// Functions/Keypoint Features/F_VN_FindReferenceKeyPointsInImageAKAZE

	{attribute 'TcIecLibraryType'}
	{attribute 'external_name' := 'F_VN_FindReferenceKeyPointsInImageAKAZE_GUID_BDEC472E_8EBA_B1D3_501C_E84D71D3DFEF'}
	(* Searches a reference image, represented by its AKAZE keypoints and corresponding descriptors, in a given source image (uses the default TcVnParamsAKAZE parameters). *)
	FUNCTION F_VN_FindReferenceKeyPointsInImageAKAZE : HRESULT
	VAR_INPUT
		ipSrcImage	:	ITcVnImage;	(* Source image *)
		ipRefKeyPoints	:	ITcVnContainer;	(* KeyPoints of the reference image, e.g. computed with F_VN_KeyPointsAndDescriptorsAKAZE (ContainerType_Vector_TcVnKeyPoint) *)
		ipRefDescriptors	:	ITcVnImage;	(* Descriptors of the reference image KeyPoints, e.g. computed with F_VN_KeyPointsAndDescriptorsAKAZE *)
		nRefImageWidth	:	UDINT;	(* Width of the reference image in pixels *)
		nRefImageHeight	:	UDINT;	(* Height of the reference image in pixels *)
		ipEdgePoints	:	REFERENCE TO ITcVnContainer;	(* Returns a container with the 4 edge points of the reference image transformed into ipSrcImage coordinates (ContainerType_Vector_TcVnPoint2_REAL) *)
		fMaxDist	:	REAL;	(* Maximum allowed descriptor distance (-1 disables this filter criterion) *)
		fMaxKnnRatio	:	REAL;	(* Maximum allowed distance ratio between first and second best match ([0..1], -1 disables this filter criterion) *)
		hrPrev	:	HRESULT;	(* HRESULT indicating the result of previous operations (If SUCCEEDED(hrPrev) equals false, no operation is executed.) *)
	END_VAR
	VAR_OUTPUT
		aPerspectiveTransform	:	TcVnMatrix3x3_LREAL;	(* Returns the perspective transformation matrix, which transforms the reference points to the source points *)
		nNumberOfGoodMatches	:	UDINT;	(* Return the number of good matches *)
		nNumberOfInliers	:	UDINT;	(* Return the number of inlier matches *)
	END_VAR

END_FUNCTION

// Functions/Keypoint Features/F_VN_KeyPointsAndDescriptorsAKAZE

	{attribute 'TcIecLibraryType'}
	{attribute 'external_name' := 'F_VN_KeyPointsAndDescriptorsAKAZE_GUID_3790B025_A52C_B22C_6EF2_34873295F067'}
	(* Detects keypoints and compute descriptors using the AKAZE method. *)
	FUNCTION F_VN_KeyPointsAndDescriptorsAKAZE : HRESULT
	VAR_INPUT
		ipSrcImage	:	ITcVnImage;	(* Source image *)
		ipKeyPoints	:	REFERENCE TO ITcVnContainer;	(* Returns a container which is filled with the keypoints (ContainerType_Vector_TcVnKeyPoint; Non-zero interface pointers are reused.) *)
		ipDescriptors	:	REFERENCE TO ITcVnImage;	(* Descriptor image (set to 0 if not required; 1 descriptor in each row; An appropriate image will be created if required.) *)
		hrPrev	:	HRESULT;	(* HRESULT indicating the result of previous operations (If SUCCEEDED(hrPrev) equals false, no operation is executed.) *)
	END_VAR

END_FUNCTION

// Functions/Keypoint Features/F_VN_FindReferenceKeyPointsInImageAKAZEExp

	{attribute 'TcIecLibraryType'}
	{attribute 'external_name' := 'F_VN_FindReferenceKeyPointsInImageAKAZEExp_GUID_5E4CFD0A_CE1D_BA8B_45D3_79DE9C5B1A21'}
	(* Searches a reference image, represented by its AKAZE keypoints and corresponding descriptors, in a given source image. (expert function) *)
	FUNCTION F_VN_FindReferenceKeyPointsInImageAKAZEExp : HRESULT
	VAR_INPUT
		ipSrcImage	:	ITcVnImage;	(* Source image *)
		ipRefKeyPoints	:	ITcVnContainer;	(* KeyPoints of the reference image, e.g. computed with F_VN_KeyPointsAndDescriptorsAKAZE (ContainerType_Vector_TcVnKeyPoint) *)
		ipRefDescriptors	:	ITcVnImage;	(* Descriptors of the reference image KeyPoints, e.g. computed with F_VN_KeyPointsAndDescriptorsAKAZE *)
		nRefImageWidth	:	UDINT;	(* Width of the reference image in pixels *)
		nRefImageHeight	:	UDINT;	(* Height of the reference image in pixels *)
		ipEdgePoints	:	REFERENCE TO ITcVnContainer;	(* Returns a container with the 4 edge points of the reference image transformed into ipSrcImage coordinates (ContainerType_Vector_TcVnPoint2_REAL) *)
		fMaxDist	:	REAL;	(* Maximum allowed descriptor distance (-1 disables this filter criterion) *)
		fMaxKnnRatio	:	REAL;	(* Maximum allowed distance ratio between first and second best match ([0..1], -1 disables this filter criterion) *)
		eNormType	:	ETcVnNormalizationType;	(* Normalization type used for descriptor matching *)
		ipSrcImageMask	:	ITcVnImage;	(* Mask to specify, where to look for keypoints in ipSrcImage (set to 0 if no mask required) *)
	END_VAR
	VAR_IN_OUT
		stAkazeParams	:	TcVnParamsAKAZE;	(* Parameters to configure the keypoint and descriptor computation for ipSrcImage (resulting descriptors must be compatible to ipRefDescriptors!) *)
	END_VAR
	VAR_INPUT
		eAlgorithm	:	ETcVnEstimationAlgorithm;	(* Estimation algorithm used for computing the perspective transformation between the two point sets *)
		fReprojThreshold	:	LREAL;	(* Maximum allowed reprojection error to treat a point pair as an inlier (only used if eAlgorithm is RANSAC, RHO) *)
		nMaxIterations	:	UDINT;	(* Maximum number of RANSAC iterations *)
		fConfidence	:	LREAL;	(* Confidence (0..1) *)
		hrPrev	:	HRESULT;	(* HRESULT indicating the result of previous operations (If SUCCEEDED(hrPrev) equals false, no operation is executed.) *)
	END_VAR
	VAR_OUTPUT
		aPerspectiveTransform	:	TcVnMatrix3x3_LREAL;	(* Returns the perspective transformation matrix, which transforms the reference points to the source points  *)
		nNumberOfGoodMatches	:	UDINT;	(* Return the number of good matches *)
		nNumberOfInliers	:	UDINT;	(* Return the number of inlier matches *)
	END_VAR

END_FUNCTION

// Functions/Keypoint Features/F_VN_FindReferenceKeyPointsInImageBRISK

	{attribute 'TcIecLibraryType'}
	{attribute 'external_name' := 'F_VN_FindReferenceKeyPointsInImageBRISK_GUID_C2D82A25_9CFE_BE26_6FAE_778E3D975A2B'}
	(* Searches a reference image, represented by its BRISK keypoints and corresponding descriptors, in a given source image (uses the default TcVnParamsBRISK parameters). *)
	FUNCTION F_VN_FindReferenceKeyPointsInImageBRISK : HRESULT
	VAR_INPUT
		ipSrcImage	:	ITcVnImage;	(* Source image *)
		ipRefKeyPoints	:	ITcVnContainer;	(* KeyPoints of the reference image, e.g. computed with F_VN_KeyPointsAndDescriptorsBRISK (ContainerType_Vector_TcVnKeyPoint) *)
		ipRefDescriptors	:	ITcVnImage;	(* Descriptors of the reference image KeyPoints, e.g. computed with F_VN_KeyPointsAndDescriptorsBRISK *)
		nRefImageWidth	:	UDINT;	(* Width of the reference image in pixels *)
		nRefImageHeight	:	UDINT;	(* Height of the reference image in pixels *)
		ipEdgePoints	:	REFERENCE TO ITcVnContainer;	(* Returns a container with the 4 edge points of the reference image transformed into ipSrcImage coordinates (ContainerType_Vector_TcVnPoint2_REAL) *)
		fMaxDist	:	REAL;	(* Maximum allowed descriptor distance (-1 disables this filter criterion) *)
		fMaxKnnRatio	:	REAL;	(* Maximum allowed distance ratio between first and second best match ([0..1], -1 disables this filter criterion) *)
		hrPrev	:	HRESULT;	(* HRESULT indicating the result of previous operations (If SUCCEEDED(hrPrev) equals false, no operation is executed.) *)
	END_VAR
	VAR_OUTPUT
		aPerspectiveTransform	:	TcVnMatrix3x3_LREAL;	(* Returns the perspective transformation matrix, which transforms the reference points to the source points  *)
		nNumberOfGoodMatches	:	UDINT;	(* Return the number of good matches *)
		nNumberOfInliers	:	UDINT;	(* Return the number of inlier matches *)
	END_VAR

END_FUNCTION

// Functions/Keypoint Features/F_VN_KeyPointsAndDescriptorsBRISK

	{attribute 'TcIecLibraryType'}
	{attribute 'external_name' := 'F_VN_KeyPointsAndDescriptorsBRISK_GUID_80ACF6A9_00E2_B47E_5EE7_B7DB54C32367'}
	(* Detects keypoints and compute descriptors using the BRISK method. *)
	FUNCTION F_VN_KeyPointsAndDescriptorsBRISK : HRESULT
	VAR_INPUT
		ipSrcImage	:	ITcVnImage;	(* Source image *)
		ipKeyPoints	:	REFERENCE TO ITcVnContainer;	(* Returns a container which is filled with the keypoints (ContainerType_Vector_TcVnKeyPoint; Non-zero interface pointers are reused.) *)
		ipDescriptors	:	REFERENCE TO ITcVnImage;	(* Descriptor image (set to 0 if not required; 1 descriptor in each row; An appropriate image will be created if required.) *)
		hrPrev	:	HRESULT;	(* HRESULT indicating the result of previous operations (If SUCCEEDED(hrPrev) equals false, no operation is executed.) *)
	END_VAR

END_FUNCTION

// Functions/Keypoint Features/F_VN_FindReferenceKeyPointsInImageBRISKExp

	{attribute 'TcIecLibraryType'}
	{attribute 'external_name' := 'F_VN_FindReferenceKeyPointsInImageBRISKExp_GUID_80D48747_D480_BAFA_427A_5CC119E86B78'}
	(* Searches a reference image, represented by its BRISK keypoints and corresponding descriptors, in a given source image. (expert function) *)
	FUNCTION F_VN_FindReferenceKeyPointsInImageBRISKExp : HRESULT
	VAR_INPUT
		ipSrcImage	:	ITcVnImage;	(* Source image *)
		ipRefKeyPoints	:	ITcVnContainer;	(* KeyPoints of the reference image, e.g. computed with F_VN_KeyPointsAndDescriptorsBRISK (ContainerType_Vector_TcVnKeyPoint) *)
		ipRefDescriptors	:	ITcVnImage;	(* Descriptors of the reference image KeyPoints, e.g. computed with F_VN_KeyPointsAndDescriptorsBRISK *)
		nRefImageWidth	:	UDINT;	(* Width of the reference image in pixels *)
		nRefImageHeight	:	UDINT;	(* Height of the reference image in pixels *)
		ipEdgePoints	:	REFERENCE TO ITcVnContainer;	(* Returns a container with the 4 edge points of the reference image transformed into ipSrcImage coordinates (ContainerType_Vector_TcVnPoint2_REAL) *)
		fMaxDist	:	REAL;	(* Maximum allowed descriptor distance (-1 disables this filter criterion) *)
		fMaxKnnRatio	:	REAL;	(* Maximum allowed distance ratio between first and second best match ([0..1], -1 disables this filter criterion) *)
		eNormType	:	ETcVnNormalizationType;	(* Normalization type used for descriptor matching *)
		ipSrcImageMask	:	ITcVnImage;	(* Mask to specify, where to look for keypoints in ipSrcImage (set to 0 if no mask required) *)
	END_VAR
	VAR_IN_OUT
		stBriskParams	:	TcVnParamsBRISK;	(* Parameters to configure the keypoint and descriptor computation for ipSrcImage (resulting descriptors must be compatible to ipRefDescriptors!) *)
	END_VAR
	VAR_INPUT
		eAlgorithm	:	ETcVnEstimationAlgorithm;	(* Estimation algorithm used for computing the perspective transformation between the two point sets *)
		fReprojThreshold	:	LREAL;	(* Maximum allowed reprojection error to treat a point pair as an inlier (only used if eAlgorithm is RANSAC, RHO) *)
		nMaxIterations	:	UDINT;	(* Maximum number of RANSAC iterations *)
		fConfidence	:	LREAL;	(* Confidence (0..1) *)
		hrPrev	:	HRESULT;	(* HRESULT indicating the result of previous operations (If SUCCEEDED(hrPrev) equals false, no operation is executed.) *)
	END_VAR
	VAR_OUTPUT
		aPerspectiveTransform	:	TcVnMatrix3x3_LREAL;	(* Returns the perspective transformation matrix, which transforms the reference points to the source points  *)
		nNumberOfGoodMatches	:	UDINT;	(* Return the number of good matches *)
		nNumberOfInliers	:	UDINT;	(* Return the number of inlier matches *)
	END_VAR

END_FUNCTION

// Functions/Keypoint Features/F_VN_FindReferenceKeyPointsInImageORB

	{attribute 'TcIecLibraryType'}
	{attribute 'external_name' := 'F_VN_FindReferenceKeyPointsInImageORB_GUID_A399F5B5_AFBB_B098_689B_67E793213C97'}
	(* Searches a reference image, represented by its ORB keypoints and corresponding descriptors, in a given source image (uses the default TcVnParamsORB parameters). *)
	FUNCTION F_VN_FindReferenceKeyPointsInImageORB : HRESULT
	VAR_INPUT
		ipSrcImage	:	ITcVnImage;	(* Source image *)
		ipRefKeyPoints	:	ITcVnContainer;	(* KeyPoints of the reference image, e.g. computed with F_VN_KeyPointsAndDescriptorsORB (ContainerType_Vector_TcVnKeyPoint) *)
		ipRefDescriptors	:	ITcVnImage;	(* Descriptors of the reference image KeyPoints, e.g. computed with F_VN_KeyPointsAndDescriptorsORB *)
		nRefImageWidth	:	UDINT;	(* Width of the reference image in pixels *)
		nRefImageHeight	:	UDINT;	(* Height of the reference image in pixels *)
		ipEdgePoints	:	REFERENCE TO ITcVnContainer;	(* Returns a container with the 4 edge points of the reference image transformed into ipSrcImage coordinates (ContainerType_Vector_TcVnPoint2_REAL) *)
		fMaxDist	:	REAL;	(* Maximum allowed descriptor distance (-1 disables this filter criterion) *)
		fMaxKnnRatio	:	REAL;	(* Maximum allowed distance ratio between first and second best match ([0..1], -1 disables this filter criterion) *)
		hrPrev	:	HRESULT;	(* HRESULT indicating the result of previous operations (If SUCCEEDED(hrPrev) equals false, no operation is executed.) *)
	END_VAR
	VAR_OUTPUT
		aPerspectiveTransform	:	TcVnMatrix3x3_LREAL;	(* Returns the perspective transformation matrix, which transforms the reference points to the source points  *)
		nNumberOfGoodMatches	:	UDINT;	(* Return the number of good matches *)
		nNumberOfInliers	:	UDINT;	(* Return the number of inlier matches *)
	END_VAR

END_FUNCTION

// Functions/Keypoint Features/F_VN_KeyPointsAndDescriptorsORB

	{attribute 'TcIecLibraryType'}
	{attribute 'external_name' := 'F_VN_KeyPointsAndDescriptorsORB_GUID_9B3AA294_CED6_B519_5EF5_95893521A0BF'}
	(* Detects keypoints and compute descriptors using the ORB method. *)
	FUNCTION F_VN_KeyPointsAndDescriptorsORB : HRESULT
	VAR_INPUT
		ipSrcImage	:	ITcVnImage;	(* Source image *)
		ipKeyPoints	:	REFERENCE TO ITcVnContainer;	(* Returns a container which is filled with the keypoints (ContainerType_Vector_TcVnKeyPoint; Non-zero interface pointers are reused.) *)
		ipDescriptors	:	REFERENCE TO ITcVnImage;	(* Descriptor image (set to 0 if not required; 1 descriptor in each row; An appropriate image will be created if required.) *)
		hrPrev	:	HRESULT;	(* HRESULT indicating the result of previous operations (If SUCCEEDED(hrPrev) equals false, no operation is executed.) *)
	END_VAR

END_FUNCTION

// Functions/Keypoint Features/F_VN_FindReferenceKeyPointsInImageORBExp

	{attribute 'TcIecLibraryType'}
	{attribute 'external_name' := 'F_VN_FindReferenceKeyPointsInImageORBExp_GUID_7E9D50DC_F5A7_BAF9_6B30_7BF62E45BB76'}
	(* Searches a reference image, represented by its ORB keypoints and corresponding descriptors, in a given source image. (expert function) *)
	FUNCTION F_VN_FindReferenceKeyPointsInImageORBExp : HRESULT
	VAR_INPUT
		ipSrcImage	:	ITcVnImage;	(* Source image *)
		ipRefKeyPoints	:	ITcVnContainer;	(* KeyPoints of the reference image, e.g. computed with F_VN_KeyPointsAndDescriptorsORB (ContainerType_Vector_TcVnKeyPoint) *)
		ipRefDescriptors	:	ITcVnImage;	(* Descriptors of the reference image KeyPoints, e.g. computed with F_VN_KeyPointsAndDescriptorsORB *)
		nRefImageWidth	:	UDINT;	(* Width of the reference image in pixels *)
		nRefImageHeight	:	UDINT;	(* Height of the reference image in pixels *)
		ipEdgePoints	:	REFERENCE TO ITcVnContainer;	(* Returns a container with the 4 edge points of the reference image transformed into ipSrcImage coordinates (ContainerType_Vector_TcVnPoint2_REAL) *)
		fMaxDist	:	REAL;	(* Maximum allowed descriptor distance (-1 disables this filter criterion) *)
		fMaxKnnRatio	:	REAL;	(* Maximum allowed distance ratio between first and second best match ([0..1], -1 disables this filter criterion) *)
		eNormType	:	ETcVnNormalizationType;	(* Normalization type used for descriptor matching (HAMMING recommended for ORB, HAMMING2 if the ORB nBriefPoints parameter is 3 or 4) *)
		ipSrcImageMask	:	ITcVnImage;	(* Mask to specify, where to look for keypoints in ipSrcImage (set to 0 if no mask required) *)
	END_VAR
	VAR_IN_OUT
		stOrbParams	:	TcVnParamsORB;	(* Parameters to configure the keypoint and descriptor computation for ipSrcImage (resulting descriptors must be compatible to ipRefDescriptors!) *)
	END_VAR
	VAR_INPUT
		eAlgorithm	:	ETcVnEstimationAlgorithm;	(* Estimation algorithm used for computing the perspective transformation between the two point sets *)
		fReprojThreshold	:	LREAL;	(* Maximum allowed reprojection error to treat a point pair as an inlier (only used if eAlgorithm is RANSAC, RHO) *)
		nMaxIterations	:	UDINT;	(* Maximum number of RANSAC iterations *)
		fConfidence	:	LREAL;	(* Confidence (0..1) *)
		hrPrev	:	HRESULT;	(* HRESULT indicating the result of previous operations (If SUCCEEDED(hrPrev) equals false, no operation is executed.) *)
	END_VAR
	VAR_OUTPUT
		aPerspectiveTransform	:	TcVnMatrix3x3_LREAL;	(* Returns the perspective transformation matrix, which transforms the reference points to the source points  *)
		nNumberOfGoodMatches	:	UDINT;	(* Return the number of good matches *)
		nNumberOfInliers	:	UDINT;	(* Return the number of inlier matches *)
	END_VAR

END_FUNCTION

// Functions/Keypoint Features/F_VN_GetMatchCoordinates

	{attribute 'TcIecLibraryType'}
	{attribute 'external_name' := 'F_VN_GetMatchCoordinates_GUID_CCE05D23_FDC1_BDD4_6441_7DE9B64CAB8C'}
	(* Return the coordinates of keypoints that match each other. *)
	FUNCTION F_VN_GetMatchCoordinates : HRESULT
	VAR_INPUT
		ipQueryKeyPoints	:	ITcVnContainer;	(* Container with query Keypoints (i.e. keypoints of a reference/template image) of type CTcVnContainer_Vector_TcVnKeyPoint *)
		ipTrainKeyPoints	:	ITcVnContainer;	(* Container with training Keypoints (i.e. keypoints of a source/input image) of type CTcVnContainer_Vector_TcVnKeyPoint *)
		ipMatches	:	ITcVnContainer;	(* Container with matches between query and train Keypoints (CTcVnContainer_Vector_TcVnDMatch). *)
		ipQueryCoordinates	:	REFERENCE TO ITcVnContainer;	(* Returns a container with the coordinates of keypoints from the query Keypoints that exist in ipMatches (CTcVnContainer_Vector_TcVnPoint2_REAL) *)
		ipTrainCoordinates	:	REFERENCE TO ITcVnContainer;	(* Returns a container with the coordinates of keypoints from the training Keypoints that exist in ipMatches (CTcVnContainer_Vector_TcVnPoint2_REAL) *)
		hrPrev	:	HRESULT;	(* HRESULT indicating the result of previous operations (If SUCCEEDED(hrPrev) equals false, no operation is executed.) *)
	END_VAR

END_FUNCTION

// Functions/Keypoint Features/F_VN_KeyPointsAGAST

	{attribute 'TcIecLibraryType'}
	{attribute 'external_name' := 'F_VN_KeyPointsAGAST_GUID_8F71829D_DD79_B116_5FE9_DE8205CB3155'}
	(* Detects keypoints using the AGAST method. *)
	FUNCTION F_VN_KeyPointsAGAST : HRESULT
	VAR_INPUT
		ipSrcImage	:	ITcVnImage;	(* Source image *)
		ipKeyPoints	:	REFERENCE TO ITcVnContainer;	(* Returns a container which is filled with the keypoints (ContainerType_Vector_TcVnKeyPoint; Non-zero interface pointers are reused.) *)
		hrPrev	:	HRESULT;	(* HRESULT indicating the result of previous operations (If SUCCEEDED(hrPrev) equals false, no operation is executed.) *)
	END_VAR

END_FUNCTION

// Functions/Keypoint Features/F_VN_KeyPointsAGASTExp

	{attribute 'TcIecLibraryType'}
	{attribute 'external_name' := 'F_VN_KeyPointsAGASTExp_GUID_980BC3B0_52B0_B73D_65D6_531BF1F1953A'}
	(* Detects keypoints using the AGAST method. (expert function) *)
	FUNCTION F_VN_KeyPointsAGASTExp : HRESULT
	VAR_INPUT
		ipSrcImage	:	ITcVnImage;	(* Source image *)
		ipKeyPoints	:	REFERENCE TO ITcVnContainer;	(* Returns a container which is filled with the keypoints (ContainerType_Vector_TcVnKeyPoint; Non-zero interface pointers are reused.) *)
		ipMask	:	ITcVnImage;	(* Mask to specify, where to look for keypoints (set to 0 if no mask required) *)
	END_VAR
	VAR_IN_OUT
		stParams	:	TcVnParamsAGAST;	(* Additional expert parameters *)
	END_VAR
	VAR_INPUT
		hrPrev	:	HRESULT;	(* HRESULT indicating the result of previous operations (If SUCCEEDED(hrPrev) equals false, no operation is executed.) *)
	END_VAR

END_FUNCTION

// Functions/Keypoint Features/F_VN_KeyPointsAndDescriptorsAKAZEExp

	{attribute 'TcIecLibraryType'}
	{attribute 'external_name' := 'F_VN_KeyPointsAndDescriptorsAKAZEExp_GUID_6F9A76DD_D14F_B87F_5276_5EACEF61BF6B'}
	(* Detects keypoints and compute descriptors using the AKAZE method. (expert function) *)
	FUNCTION F_VN_KeyPointsAndDescriptorsAKAZEExp : HRESULT
	VAR_INPUT
		ipSrcImage	:	ITcVnImage;	(* Source image *)
		ipKeyPoints	:	REFERENCE TO ITcVnContainer;	(* Returns a container which is filled with the keypoints (ContainerType_Vector_TcVnKeyPoint; Non-zero interface pointers are reused.) *)
		ipDescriptors	:	REFERENCE TO ITcVnImage;	(* Descriptor image (set to 0 if not required; 1 descriptor in each row; An appropriate image will be created if required.) *)
		ipMask	:	ITcVnImage;	(* Mask to specify, where to look for keypoints (set to 0 if no mask required) *)
	END_VAR
	VAR_IN_OUT
		stParams	:	TcVnParamsAKAZE;	(* Additional expert parameters *)
	END_VAR
	VAR_INPUT
		hrPrev	:	HRESULT;	(* HRESULT indicating the result of previous operations (If SUCCEEDED(hrPrev) equals false, no operation is executed.) *)
	END_VAR

END_FUNCTION

// Functions/Keypoint Features/F_VN_KeyPointsAndDescriptorsBRISKExp

	{attribute 'TcIecLibraryType'}
	{attribute 'external_name' := 'F_VN_KeyPointsAndDescriptorsBRISKExp_GUID_DE018668_62DF_B383_7088_5E0B7EA37FE7'}
	(* Detects keypoints and compute descriptors using the BRISK method. (expert function) *)
	FUNCTION F_VN_KeyPointsAndDescriptorsBRISKExp : HRESULT
	VAR_INPUT
		ipSrcImage	:	ITcVnImage;	(* Source image *)
		ipKeyPoints	:	REFERENCE TO ITcVnContainer;	(* Returns a container which is filled with the keypoints (ContainerType_Vector_TcVnKeyPoint; Non-zero interface pointers are reused.) *)
		ipDescriptors	:	REFERENCE TO ITcVnImage;	(* Descriptor image (set to 0 if not required; 1 descriptor in each row; An appropriate image will be created if required.) *)
		ipMask	:	ITcVnImage;	(* Mask to specify, where to look for keypoints (set to 0 if no mask required) *)
	END_VAR
	VAR_IN_OUT
		stParams	:	TcVnParamsBRISK;	(* Additional expert parameters *)
	END_VAR
	VAR_INPUT
		hrPrev	:	HRESULT;	(* HRESULT indicating the result of previous operations (If SUCCEEDED(hrPrev) equals false, no operation is executed.) *)
	END_VAR

END_FUNCTION

// Functions/Keypoint Features/F_VN_KeyPointsAndDescriptorsKAZE

	{attribute 'TcIecLibraryType'}
	{attribute 'external_name' := 'F_VN_KeyPointsAndDescriptorsKAZE_GUID_CF12748A_0DA3_BE86_6DFA_1901CBB9FB17'}
	(* Detects keypoints and compute descriptors using the KAZE method. *)
	FUNCTION F_VN_KeyPointsAndDescriptorsKAZE : HRESULT
	VAR_INPUT
		ipSrcImage	:	ITcVnImage;	(* Source image *)
		ipKeyPoints	:	REFERENCE TO ITcVnContainer;	(* Returns a container which is filled with the keypoints (ContainerType_Vector_TcVnKeyPoint; Non-zero interface pointers are reused.) *)
		ipDescriptors	:	REFERENCE TO ITcVnImage;	(* Descriptor image (set to 0 if not required; 1 descriptor in each row; An appropriate image will be created if required.) *)
		hrPrev	:	HRESULT;	(* HRESULT indicating the result of previous operations (If SUCCEEDED(hrPrev) equals false, no operation is executed.) *)
	END_VAR

END_FUNCTION

// Functions/Keypoint Features/F_VN_KeyPointsAndDescriptorsKAZEExp

	{attribute 'TcIecLibraryType'}
	{attribute 'external_name' := 'F_VN_KeyPointsAndDescriptorsKAZEExp_GUID_AFA123DE_6B39_B2E5_7E54_59838DFABED7'}
	(* Detects keypoints and compute descriptors using the KAZE method. (expert function) *)
	FUNCTION F_VN_KeyPointsAndDescriptorsKAZEExp : HRESULT
	VAR_INPUT
		ipSrcImage	:	ITcVnImage;	(* Source image *)
		ipKeyPoints	:	REFERENCE TO ITcVnContainer;	(* Returns a container which is filled with the keypoints (ContainerType_Vector_TcVnKeyPoint; Non-zero interface pointers are reused.) *)
		ipDescriptors	:	REFERENCE TO ITcVnImage;	(* Descriptor image (set to 0 if not required; 1 descriptor in each row; An appropriate image will be created if required.) *)
		ipMask	:	ITcVnImage;	(* Mask to specify, where to look for keypoints (set to 0 if no mask required) *)
	END_VAR
	VAR_IN_OUT
		stParams	:	TcVnParamsKAZE;	(* Additional expert parameters *)
	END_VAR
	VAR_INPUT
		hrPrev	:	HRESULT;	(* HRESULT indicating the result of previous operations (If SUCCEEDED(hrPrev) equals false, no operation is executed.) *)
	END_VAR

END_FUNCTION

// Functions/Keypoint Features/F_VN_KeyPointsAndDescriptorsORBExp

	{attribute 'TcIecLibraryType'}
	{attribute 'external_name' := 'F_VN_KeyPointsAndDescriptorsORBExp_GUID_E6A25B2C_BB26_BD0B_7FD0_3740AF141B87'}
	(* Detect keypoints and compute descriptors using the ORB method. (expert function) *)
	FUNCTION F_VN_KeyPointsAndDescriptorsORBExp : HRESULT
	VAR_INPUT
		ipSrcImage	:	ITcVnImage;	(* Source image *)
		ipKeyPoints	:	REFERENCE TO ITcVnContainer;	(* Returns a container which is filled with the keypoints (ContainerType_Vector_TcVnKeyPoint; Non-zero interface pointers are reused.) *)
		ipDescriptors	:	REFERENCE TO ITcVnImage;	(* Descriptor image (set to 0 if not required; 1 descriptor in each row; An appropriate image will be created if required.) *)
		ipMask	:	ITcVnImage;	(* Mask to specify, where to look for keypoints (set to 0 if no mask required) *)
	END_VAR
	VAR_IN_OUT
		stParams	:	TcVnParamsORB;	(* Additional expert parameters *)
	END_VAR
	VAR_INPUT
		hrPrev	:	HRESULT;	(* HRESULT indicating the result of previous operations (If SUCCEEDED(hrPrev) equals false, no operation is executed.) *)
	END_VAR

END_FUNCTION

// Functions/Keypoint Features/F_VN_KeyPointsFAST

	{attribute 'TcIecLibraryType'}
	{attribute 'external_name' := 'F_VN_KeyPointsFAST_GUID_57AACB9F_2688_BD91_5750_FD570F10A14B'}
	(* Detects keypoints using the FAST method. *)
	FUNCTION F_VN_KeyPointsFAST : HRESULT
	VAR_INPUT
		ipSrcImage	:	ITcVnImage;	(* Source image (single-channel). *)
		ipKeyPoints	:	REFERENCE TO ITcVnContainer;	(* Returns a container which is filled with the keypoints (ContainerType_Vector_TcVnKeyPoint; Non-zero interface pointers are reused.) *)
		hrPrev	:	HRESULT;	(* HRESULT indicating the result of previous operations (If SUCCEEDED(hrPrev) equals false, no operation is executed.) *)
	END_VAR

END_FUNCTION

// Functions/Keypoint Features/F_VN_KeyPointsFASTExp

	{attribute 'TcIecLibraryType'}
	{attribute 'external_name' := 'F_VN_KeyPointsFASTExp_GUID_8D7068F4_30C2_BA25_489C_91A7586E80BE'}
	(* Detects keypoints using the FAST method. (expert function) *)
	FUNCTION F_VN_KeyPointsFASTExp : HRESULT
	VAR_INPUT
		ipSrcImage	:	ITcVnImage;	(* Source image *)
		ipKeyPoints	:	REFERENCE TO ITcVnContainer;	(* Returns a container which is filled with the keypoints (ContainerType_Vector_TcVnKeyPoint; Non-zero interface pointers are reused.) *)
		ipMask	:	ITcVnImage;	(* Mask to specify, where to look for keypoints (set to 0 if no mask required) *)
	END_VAR
	VAR_IN_OUT
		stParams	:	TcVnParamsFAST;	(* Additional expert parameters *)
	END_VAR
	VAR_INPUT
		hrPrev	:	HRESULT;	(* HRESULT indicating the result of previous operations (If SUCCEEDED(hrPrev) equals false, no operation is executed.) *)
	END_VAR

END_FUNCTION

// Functions/Keypoint Features/F_VN_KeyPointsGFTT

	{attribute 'TcIecLibraryType'}
	{attribute 'external_name' := 'F_VN_KeyPointsGFTT_GUID_4F2F2F01_B101_B8F2_69C0_E95BDCC4F7CF'}
	(* Detects keypoints using the GFTT method, which detects strong corners. *)
	FUNCTION F_VN_KeyPointsGFTT : HRESULT
	VAR_INPUT
		ipSrcImage	:	ITcVnImage;	(* Source image *)
		ipKeyPoints	:	REFERENCE TO ITcVnContainer;	(* Returns a container which is filled with the keypoints (ContainerType_Vector_TcVnKeyPoint; Non-zero interface pointers are reused.) *)
		hrPrev	:	HRESULT;	(* HRESULT indicating the result of previous operations (If SUCCEEDED(hrPrev) equals false, no operation is executed.) *)
	END_VAR

END_FUNCTION

// Functions/Keypoint Features/F_VN_KeyPointsGFTTExp

	{attribute 'TcIecLibraryType'}
	{attribute 'external_name' := 'F_VN_KeyPointsGFTTExp_GUID_C3513AC9_42DF_BA18_716F_91B2FD8F288E'}
	(* Detects keypoints using the GFTT method, which detects strong corners. (expert function) *)
	FUNCTION F_VN_KeyPointsGFTTExp : HRESULT
	VAR_INPUT
		ipSrcImage	:	ITcVnImage;	(* Source image *)
		ipKeyPoints	:	REFERENCE TO ITcVnContainer;	(* Returns a container which is filled with the keypoints (ContainerType_Vector_TcVnKeyPoint; Non-zero interface pointers are reused.) *)
		ipMask	:	ITcVnImage;	(* Mask to specify, where to look for keypoints (set to 0 if no mask required) *)
	END_VAR
	VAR_IN_OUT
		stParams	:	TcVnParamsGFTT;	(* Additional expert parameters *)
	END_VAR
	VAR_INPUT
		hrPrev	:	HRESULT;	(* HRESULT indicating the result of previous operations (If SUCCEEDED(hrPrev) equals false, no operation is executed.) *)
	END_VAR

END_FUNCTION

// Functions/Keypoint Features/F_VN_KeyPointsMSER

	{attribute 'TcIecLibraryType'}
	{attribute 'external_name' := 'F_VN_KeyPointsMSER_GUID_3109C890_21B5_B063_6136_0A0A5FE7AD58'}
	(* Detects keypoints using the MSER method. *)
	FUNCTION F_VN_KeyPointsMSER : HRESULT
	VAR_INPUT
		ipSrcImage	:	ITcVnImage;	(* Source image *)
		ipKeyPoints	:	REFERENCE TO ITcVnContainer;	(* Returns a container which is filled with the keypoints (ContainerType_Vector_TcVnKeyPoint; Non-zero interface pointers are reused.) *)
		hrPrev	:	HRESULT;	(* HRESULT indicating the result of previous operations (If SUCCEEDED(hrPrev) equals false, no operation is executed.) *)
	END_VAR

END_FUNCTION

// Functions/Keypoint Features/F_VN_KeyPointsMSERExp

	{attribute 'TcIecLibraryType'}
	{attribute 'external_name' := 'F_VN_KeyPointsMSERExp_GUID_C3D69AC4_93EC_BF69_5853_BACBB207FD71'}
	(* Detects keypoints using the MSER method. (expert function) *)
	FUNCTION F_VN_KeyPointsMSERExp : HRESULT
	VAR_INPUT
		ipSrcImage	:	ITcVnImage;	(* Source image *)
		ipKeyPoints	:	REFERENCE TO ITcVnContainer;	(* Returns a container which is filled with the keypoints (ContainerType_Vector_TcVnKeyPoint; Non-zero interface pointers are reused.) *)
		ipMask	:	ITcVnImage;	(* Mask to specify, where to look for keypoints (set to 0 if no mask required) *)
	END_VAR
	VAR_IN_OUT
		stParams	:	TcVnParamsMSER;	(* Additional expert parameters *)
	END_VAR
	VAR_INPUT
		hrPrev	:	HRESULT;	(* HRESULT indicating the result of previous operations (If SUCCEEDED(hrPrev) equals false, no operation is executed.) *)
	END_VAR

END_FUNCTION

// Functions/Keypoint Features/F_VN_KeyPointsSB

	{attribute 'TcIecLibraryType'}
	{attribute 'external_name' := 'F_VN_KeyPointsSB_GUID_42C47F1D_89C2_B76B_4125_BC63BADCF1B8'}
	(* Detects keypoints using a Simple Blob method
          - several iterations apply different thresholds to source image
          - connected components (blobs) are detected
          - the center and radius of the blobs are returned as keypoints *)
	FUNCTION F_VN_KeyPointsSB : HRESULT
	VAR_INPUT
		ipSrcImage	:	ITcVnImage;	(* Source image *)
		ipKeyPoints	:	REFERENCE TO ITcVnContainer;	(* Returns a container which is filled with the keypoints (ContainerType_Vector_TcVnKeyPoint; Non-zero interface pointers are reused.) *)
		hrPrev	:	HRESULT;	(* HRESULT indicating the result of previous operations (If SUCCEEDED(hrPrev) equals false, no operation is executed.) *)
	END_VAR

END_FUNCTION

// Functions/Keypoint Features/F_VN_KeyPointsSBExp

	{attribute 'TcIecLibraryType'}
	{attribute 'external_name' := 'F_VN_KeyPointsSBExp_GUID_E9C0C92B_60E8_BE5A_5624_76F2BED69B6B'}
	(* Detects keypoints using a Simple Blob method (expert function)
          - several iterations apply different thresholds to source image
          - connected components (blobs) are detected
          - the center and radius of the blobs are returned as keypoints *)
	FUNCTION F_VN_KeyPointsSBExp : HRESULT
	VAR_INPUT
		ipSrcImage	:	ITcVnImage;	(* Source image *)
		ipKeyPoints	:	REFERENCE TO ITcVnContainer;	(* Returns a container which is filled with the keypoints (ContainerType_Vector_TcVnKeyPoint; Non-zero interface pointers are reused.) *)
		ipMask	:	ITcVnImage;	(* Mask to specify, where to look for keypoints (optional, set to 0 if not required) *)
	END_VAR
	VAR_IN_OUT
		stParams	:	TcVnParamsSB;	(* Several parameters to filter the detected blobs *)
	END_VAR
	VAR_INPUT
		hrPrev	:	HRESULT;	(* HRESULT indicating the result of previous operations (If SUCCEEDED(hrPrev) equals false, no operation is executed.) *)
	END_VAR

END_FUNCTION

// Functions/Keypoint Features/F_VN_MatchDescriptorsBF

	{attribute 'TcIecLibraryType'}
	{attribute 'external_name' := 'F_VN_MatchDescriptorsBF_GUID_DBA2D75F_1932_BE9B_4D81_03D5A0C41A44'}
	(* Match descriptors using a brute force approach. *)
	FUNCTION F_VN_MatchDescriptorsBF : HRESULT
	VAR_INPUT
		ipQueryDescriptors	:	ITcVnImage;	(* Query descriptors (i.e. descriptors of a reference/template image) *)
		ipTrainDescriptors	:	ITcVnImage;	(* Training descriptors (i.e. descriptors of a source/input image) *)
		ipMatches	:	REFERENCE TO ITcVnContainer;	(* Returns a container which is filled with the descriptor matches (ContainerType_Vector_TcVnDMatch; Non-zero interface pointers are reused.) *)
		hrPrev	:	HRESULT;	(* HRESULT indicating the result of previous operations (If SUCCEEDED(hrPrev) equals false, no operation is executed.) *)
	END_VAR

END_FUNCTION

// Functions/Keypoint Features/F_VN_MatchDescriptorsBFExp

	{attribute 'TcIecLibraryType'}
	{attribute 'external_name' := 'F_VN_MatchDescriptorsBFExp_GUID_2AB78C3E_9D7D_B432_7622_3B8E95EFE658'}
	(* Match descriptors using a brute force approach. (expert function) *)
	FUNCTION F_VN_MatchDescriptorsBFExp : HRESULT
	VAR_INPUT
		ipQueryDescriptors	:	ITcVnImage;	(* Query descriptors (i.e. descriptors of a reference/template image) *)
		ipTrainDescriptors	:	ITcVnImage;	(* Training descriptors (i.e. descriptors of a source/input image) *)
		ipMatches	:	REFERENCE TO ITcVnContainer;	(* Returns a container which is filled with the descriptor matches (ContainerType_Vector_TcVnDMatch; Non-zero interface pointers are reused.) *)
		ipMask	:	ITcVnImage;	(* Mask to specify permissable matches, i.e. query[i] can be matched with train[j] only if mask[i][j] != 0 (set to 0 if no mask required) *)
		eNormType	:	ETcVnNormalizationType;	(* Normalization type (only L1, L2, L2SQR, HAMMING, HAMMING2 supported). HAMMING2 should be used for ORB descriptors if the ORB nBriefPoints parameter is 3 or 4) *)
		bCrossCheck	:	BOOL;	(* If true, only consistent matches are returned, i.e. query->train and train->query detect the same match *)
		hrPrev	:	HRESULT;	(* HRESULT indicating the result of previous operations (If SUCCEEDED(hrPrev) equals false, no operation is executed.) *)
	END_VAR

END_FUNCTION

// Functions/Keypoint Features/F_VN_MatchDescriptorsFlannLsh

	{attribute 'TcIecLibraryType'}
	{attribute 'external_name' := 'F_VN_MatchDescriptorsFlannLsh_GUID_023CD41D_1F3A_B6B3_6D2F_7791E7D7382A'}
	(* Match descriptors using a FLANN based approach with LSH index. *)
	FUNCTION F_VN_MatchDescriptorsFlannLsh : HRESULT
	VAR_INPUT
		ipQueryDescriptors	:	ITcVnImage;	(* Query descriptors (i.e. descriptors of a reference/template image) *)
		ipTrainDescriptors	:	ITcVnImage;	(* Training descriptors (i.e. descriptors of a source/input image) *)
		ipMatches	:	REFERENCE TO ITcVnContainer;	(* Returns a container which is filled with the descriptor matches (ContainerType_Vector_TcVnDMatch; Non-zero interface pointers are reused.) *)
		hrPrev	:	HRESULT;	(* HRESULT indicating the result of previous operations (If SUCCEEDED(hrPrev) equals false, no operation is executed.) *)
	END_VAR

END_FUNCTION

// Functions/Keypoint Features/F_VN_MatchDescriptorsFlannLshExp

	{attribute 'TcIecLibraryType'}
	{attribute 'external_name' := 'F_VN_MatchDescriptorsFlannLshExp_GUID_CE80D858_FCA0_B75E_7AC8_1C42533236A1'}
	(* Match descriptors using a FLANN based approach with LSH index. (expert function) *)
	FUNCTION F_VN_MatchDescriptorsFlannLshExp : HRESULT
	VAR_INPUT
		ipQueryDescriptors	:	ITcVnImage;	(* Query descriptors (i.e. descriptors of a reference/template image) *)
		ipTrainDescriptors	:	ITcVnImage;	(* Training descriptors (i.e. descriptors of a source/input image) *)
		ipMatches	:	REFERENCE TO ITcVnContainer;	(* Returns a container which is filled with the descriptor matches (ContainerType_Vector_TcVnDMatch; Non-zero interface pointers are reused.) *)
		nTableNumber	:	UDINT;	(* Number of tables *)
		nKeySize	:	UDINT;	(* Key size *)
		nMultiProbeLevel	:	UDINT;	(* Multi-probe level *)
		nChecks	:	UDINT;	(* Maximum number of visited leafs when searching for neighbors *)
		hrPrev	:	HRESULT;	(* HRESULT indicating the result of previous operations (If SUCCEEDED(hrPrev) equals false, no operation is executed.) *)
	END_VAR

END_FUNCTION

// Functions/Keypoint Features/F_VN_MatchDescriptorsKnnBF

	{attribute 'TcIecLibraryType'}
	{attribute 'external_name' := 'F_VN_MatchDescriptorsKnnBF_GUID_6B1CF23F_0905_B925_456A_231D87908FC0'}
	(* Match descriptors (k nearest neighbors) using a brute force approach. *)
	FUNCTION F_VN_MatchDescriptorsKnnBF : HRESULT
	VAR_INPUT
		ipQueryDescriptors	:	ITcVnImage;	(* Query descriptors (i.e. descriptors of a reference/template image) *)
		ipTrainDescriptors	:	ITcVnImage;	(* Training descriptors (i.e. descriptors of a source/input image) *)
		ipMatches	:	REFERENCE TO ITcVnContainer;	(* Returns a container which is filled with the descriptor matches (ContainerType_Vector_Vector_TcVnDMatch; Non-zero interface pointers are reused.) *)
		nK	:	UDINT;	(* Number of required best train matches for each query descriptor (i.e. nk := 2) *)
		hrPrev	:	HRESULT;	(* HRESULT indicating the result of previous operations (If SUCCEEDED(hrPrev) equals false, no operation is executed.) *)
	END_VAR

END_FUNCTION

// Functions/Keypoint Features/F_VN_MatchDescriptorsKnnBFExp

	{attribute 'TcIecLibraryType'}
	{attribute 'external_name' := 'F_VN_MatchDescriptorsKnnBFExp_GUID_276BF34B_EFF3_B225_7DF9_9A06B02FBED4'}
	(* Match descriptors (k nearest neighbors) using a brute force approach. (expert function) *)
	FUNCTION F_VN_MatchDescriptorsKnnBFExp : HRESULT
	VAR_INPUT
		ipQueryDescriptors	:	ITcVnImage;	(* Query descriptors (i.e. descriptors of a reference/template image) *)
		ipTrainDescriptors	:	ITcVnImage;	(* Training descriptors (i.e. descriptors of a source/input image) *)
		ipMatches	:	REFERENCE TO ITcVnContainer;	(* Returns a container which is filled with the descriptor matches (ContainerType_Vector_Vector_TcVnDMatch; Non-zero interface pointers are reused.) *)
		nK	:	UDINT;	(* Number of required best train matches for each query descriptor (i.e. nk := 2) *)
		ipMask	:	ITcVnImage;	(* Mask to specify permissable matches, i.e. query[i] can be matched with train[j] only if mask[i][j] != 0 (set to 0 if no mask required) *)
		bCompactResult	:	BOOL;	(* If true, matches vector does not contain entries for fully masked-out query descriptors *)
		eNormType	:	ETcVnNormalizationType;	(* Normalization type (only L1, L2, L2SQR, HAMMING, HAMMING2 supported). HAMMING2 should be used for ORB descriptors if the ORB nBriefPoints parameter is 3 or 4) *)
		bCrossCheck	:	BOOL;	(* If true, only consistent matches are returned, i.e. query->train and train->query detect the same match (only used if nK = 1) *)
		hrPrev	:	HRESULT;	(* HRESULT indicating the result of previous operations (If SUCCEEDED(hrPrev) equals false, no operation is executed.) *)
	END_VAR

END_FUNCTION

// Functions/Keypoint Features/F_VN_MatchDescriptorsKnnFlannLsh

	{attribute 'TcIecLibraryType'}
	{attribute 'external_name' := 'F_VN_MatchDescriptorsKnnFlannLsh_GUID_A010F6AD_66F9_B954_4B43_138EF271714F'}
	(* Match descriptors (k nearest neighbors) using a FLANN based approach with LSH index. *)
	FUNCTION F_VN_MatchDescriptorsKnnFlannLsh : HRESULT
	VAR_INPUT
		ipQueryDescriptors	:	ITcVnImage;	(* Query descriptors (i.e. descriptors of a reference/template image) *)
		ipTrainDescriptors	:	ITcVnImage;	(* Training descriptors (i.e. descriptors of a source/input image) *)
		ipMatches	:	REFERENCE TO ITcVnContainer;	(* Returns a container which is filled with the descriptor matches (ContainerType_Vector_Vector_TcVnDMatch; Non-zero interface pointers are reused.) *)
		nK	:	UDINT;	(* Number of required best train matches for each query descriptor (i.e. nk := 2) *)
		hrPrev	:	HRESULT;	(* HRESULT indicating the result of previous operations (If SUCCEEDED(hrPrev) equals false, no operation is executed.) *)
	END_VAR

END_FUNCTION

// Functions/Keypoint Features/F_VN_MatchDescriptorsKnnFlannLshExp

	{attribute 'TcIecLibraryType'}
	{attribute 'external_name' := 'F_VN_MatchDescriptorsKnnFlannLshExp_GUID_ACA8AE96_2D7B_B935_5617_06D2724DA717'}
	(* Match descriptors (k nearest neighbors) using a FLANN based approach with LSH index. (expert function) *)
	FUNCTION F_VN_MatchDescriptorsKnnFlannLshExp : HRESULT
	VAR_INPUT
		ipQueryDescriptors	:	ITcVnImage;	(* Query descriptors (i.e. descriptors of a reference/template image) *)
		ipTrainDescriptors	:	ITcVnImage;	(* Training descriptors (i.e. descriptors of a source/input image) *)
		ipMatches	:	REFERENCE TO ITcVnContainer;	(* Returns a container which is filled with the descriptor matches (ContainerType_Vector_Vector_TcVnDMatch; Non-zero interface pointers are reused.) *)
		nK	:	UDINT;	(* Number of required best train matches for each query descriptor (i.e. nk := 2) *)
		nTableNumber	:	UDINT;	(* Number of tables *)
		nKeySize	:	UDINT;	(* Key size *)
		nMultiProbeLevel	:	UDINT;	(* Multi-probe level *)
		nChecks	:	UDINT;	(* Maximum number of visited leafs when searching for neighbors *)
		hrPrev	:	HRESULT;	(* HRESULT indicating the result of previous operations (If SUCCEEDED(hrPrev) equals false, no operation is executed.) *)
	END_VAR

END_FUNCTION

// Functions/Keypoint Features/F_VN_RegionsMSER

	{attribute 'TcIecLibraryType'}
	{attribute 'external_name' := 'F_VN_RegionsMSER_GUID_3D40AB9C_52E4_B914_52DC_C3D7F66C36C0'}
	(* Detects regions using the MSER method. *)
	FUNCTION F_VN_RegionsMSER : HRESULT
	VAR_INPUT
		ipSrcImage	:	ITcVnImage;	(* Source image *)
		ipRegions	:	REFERENCE TO ITcVnContainer;	(* Returns a container which is filled with the region points (ContainerType_Vector_Vector_TcVnPoint2_DINT; Non-zero interface pointers are reused.) *)
		ipBoundingBoxes	:	REFERENCE TO ITcVnContainer;	(* Returns a container which is filled with the region bounding boxes (ContainerType_Vector_TcVnRectangle_DINT; Non-zero interface pointers are reused.) *)
		hrPrev	:	HRESULT;	(* HRESULT indicating the result of previous operations (If SUCCEEDED(hrPrev) equals false, no operation is executed.) *)
	END_VAR

END_FUNCTION

// Functions/Keypoint Features/F_VN_RegionsMSERExp

	{attribute 'TcIecLibraryType'}
	{attribute 'external_name' := 'F_VN_RegionsMSERExp_GUID_8CBCCE29_857B_B7C8_73FE_BADCD47BF7B7'}
	(* Detects regions using the MSER method. (expert function) *)
	FUNCTION F_VN_RegionsMSERExp : HRESULT
	VAR_INPUT
		ipSrcImage	:	ITcVnImage;	(* Source image *)
		ipRegions	:	REFERENCE TO ITcVnContainer;	(* Returns a container which is filled with the region points (ContainerType_Vector_Vector_TcVnPoint2_DINT; Non-zero interface pointers are reused.) *)
		ipBoundingBoxes	:	REFERENCE TO ITcVnContainer;	(* Returns a container which is filled with the region bounding boxes (ContainerType_Vector_TcVnRectangle_DINT; Non-zero interface pointers are reused.) *)
	END_VAR
	VAR_IN_OUT
		stParams	:	TcVnParamsMSER;	(* Additional expert parameters *)
	END_VAR
	VAR_INPUT
		hrPrev	:	HRESULT;	(* HRESULT indicating the result of previous operations (If SUCCEEDED(hrPrev) equals false, no operation is executed.) *)
	END_VAR

END_FUNCTION

// Functions/Code Quality/F_VN_GradeBarcode

	{attribute 'TcIecLibraryType'}
	{attribute 'external_name' := 'F_VN_GradeBarcode_GUID_11D0B735_4CF7_B3D6_4EF9_B2D212E4DFBC'}
	(* Grades a 1D barcode according to ISO / IEC 15416:2016. Requires uniform illumination, good focus and the image sensor plane parallel to the code plane to achieve meaningful results. *)
	FUNCTION F_VN_GradeBarcode : HRESULT
	VAR_INPUT
		ipSrcImage	:	ITcVnImage;	(* Source image, only containing the horizontally aligned barcode region (USINT, 1 channel, including quiet zones on left and right, excluding Text or empty space on more than 10% total height on top or bottom) *)
		ipDecodedData	:	REFERENCE TO ITcVnContainer;	(* Returns the decoded data (ContainerType_String_SINT) *)
	END_VAR
	VAR_IN_OUT
		stCodeGrades	:	TcVnCodeGrades1D;	(* Returns the code grades in the range from 0 (very bad) to 4 (very good) *)
	END_VAR
	VAR_INPUT
		eBarcodeType	:	ETcVnBarcodeType;	(* Type of the barcode (supported: CODE39, CODE128, EAN8, EAN13, ITF, UPCA, UPCE) *)
		hrPrev	:	HRESULT;	(* HRESULT indicating the result of previous operations (If SUCCEEDED(hrPrev) equals false, no operation is executed.) *)
	END_VAR
	VAR_OUTPUT
		fAngleDeg	:	REAL;	(* Returns the approximate clockwise rotation angle in degree *)
	END_VAR

END_FUNCTION

// Functions/Code Quality/F_VN_GradeBarcodeExp

	{attribute 'TcIecLibraryType'}
	{attribute 'external_name' := 'F_VN_GradeBarcodeExp_GUID_9801F9A0_D5A6_BDF6_43B2_4057FAE04856'}
	(* Grades a 1D barcode according to ISO / IEC 15416:2016. Requires uniform illumination, good focus and the image sensor plane parallel to the code plane to achieve meaningful results. (expert function) *)
	FUNCTION F_VN_GradeBarcodeExp : HRESULT
	VAR_INPUT
		ipSrcImage	:	ITcVnImage;	(* Source image, only containing the horizontally aligned barcode region (USINT, 1 channel, including quiet zones on left and right, excluding Text or empty space on more than 10% total height on top or bottom) *)
		ipDecodedData	:	REFERENCE TO ITcVnContainer;	(* Returns the decoded data (ContainerType_String_SINT) *)
	END_VAR
	VAR_IN_OUT
		stCodeGrades	:	TcVnCodeGrades1D;	(* Returns the code grades in the range from 0 (very bad) to 4 (very good) *)
	END_VAR
	VAR_INPUT
		eBarcodeType	:	ETcVnBarcodeType;	(* Type of the barcode (supported: CODE39, CODE128, EAN8, EAN13, ITF, UPCA, UPCE) *)
		eSearchDirection	:	ETcVnBarcodeSearchDirection;	(* Barcode search direction (BSD_ANY first tries horizontal, then vertical) *)
		ipResultVisualization	:	REFERENCE TO ITcVnImage;	(* Returns a visualization of the scan lines (optional, set to 0 if not required). Grades are color coded: >= 3 as green, >= 2 as light blue, >= 1 as orange, < 1 as red *)
		ipScanLineInfo	:	REFERENCE TO ITcVnContainer;	(* Returns additional scan line info for further evaluation, e.g. to use PlotIntensityProfile for visualization (optional, set to 0 if not required; ContainerType_Vector_TcVnVector3_REAL, containing [row index, overall grade, threshold]) *)
		ipContour	:	REFERENCE TO ITcVnContainer;	(* Returns the 4 approximate code corner points, including the quiet zone (optional, set to 0 if not required; ContainerType_Vector_TcVnPoint2_DINT) *)
		hrPrev	:	HRESULT;	(* HRESULT indicating the result of previous operations (If SUCCEEDED(hrPrev) equals false, no operation is executed.) *)
	END_VAR
	VAR_OUTPUT
		fAngleDeg	:	REAL;	(* Returns the approximate clockwise rotation angle in degree *)
	END_VAR

END_FUNCTION

// Functions/Code Quality/F_VN_GradeDataMatrixCode

	{attribute 'TcIecLibraryType'}
	{attribute 'external_name' := 'F_VN_GradeDataMatrixCode_GUID_30570790_AC72_B0A0_4167_CB1726B10D10'}
	(* Grades a Data Matrix code (ECC200) according to ISO / IEC 15415:2011. Requires uniform illumination, good focus and the image sensor plane parallel to the code plane to achieve meaningful results. *)
	FUNCTION F_VN_GradeDataMatrixCode : HRESULT
	VAR_INPUT
		ipSrcImage	:	ITcVnImage;	(* Source image, only containing the Data Matrix code region (USINT, 1 channel, including quiet zone) *)
		ipDecodedData	:	REFERENCE TO ITcVnContainer;	(* Returns the decoded data (ContainerType_String_SINT) *)
	END_VAR
	VAR_IN_OUT
		stCodeGrades	:	TcVnCodeGradesDM;	(* Returns the code grades in the range from 0 (very bad) to 4 (very good) *)
	END_VAR
	VAR_INPUT
		fModuleWidth	:	REAL;	(* Minimum module width of the code in the image (in pixels). Must be at least 3, preferably 5 - 8. *)
		hrPrev	:	HRESULT;	(* HRESULT indicating the result of previous operations (If SUCCEEDED(hrPrev) equals false, no operation is executed.) *)
	END_VAR
	VAR_OUTPUT
		fAngleDeg	:	REAL;	(* Returns the clockwise rotation angle in degree *)
	END_VAR

END_FUNCTION

// Functions/Code Quality/F_VN_GradeDataMatrixCodeExp

	{attribute 'TcIecLibraryType'}
	{attribute 'external_name' := 'F_VN_GradeDataMatrixCodeExp_GUID_D33533C5_F838_B70E_7CFC_3BF84FEE0BC2'}
	(* Grades a Data Matrix code (ECC200) according to ISO / IEC 15415:2011. Requires uniform illumination, good focus and the image sensor plane parallel to the code plane to achieve meaningful results. (expert function) *)
	FUNCTION F_VN_GradeDataMatrixCodeExp : HRESULT
	VAR_INPUT
		ipSrcImage	:	ITcVnImage;	(* Source image, only containing the Data Matrix code region (USINT, 1 channel, including quiet zone) *)
		ipDecodedData	:	REFERENCE TO ITcVnContainer;	(* Returns the decoded data (ContainerType_String_SINT) *)
	END_VAR
	VAR_IN_OUT
		stCodeGrades	:	TcVnCodeGradesDM;	(* Returns the code grades in the range from 0 (very bad) to 4 (very good) *)
	END_VAR
	VAR_INPUT
		fModuleWidth	:	REAL;	(* Minimum module width of the code in the image (in pixels). Must be at least 3, preferably 5 - 8. *)
		ipResultVisualization	:	REFERENCE TO ITcVnImage;	(* Returns a visualization of the scan grid (optional, set to 0 if not required). Module margin grades are color coded: >= 3 as green, >= 2 as light blue, >= 1 as orange, < 1 as red *)
		ipMarginGrades	:	REFERENCE TO ITcVnContainer;	(* Returns the individual margin grade for each module, e.g. to create a custom visualization (optional, set to 0 if not required; ContainerType_Vector_TcVnVector3_REAL, containing [x-position, y-position, grade]) *)
		ipContour	:	REFERENCE TO ITcVnContainer;	(* Returns the 4 code corner points, excluding the quiet zone (optional, set to 0 if not required; ContainerType_Vector_TcVnPoint2_DINT) *)
		hrPrev	:	HRESULT;	(* HRESULT indicating the result of previous operations (If SUCCEEDED(hrPrev) equals false, no operation is executed.) *)
	END_VAR
	VAR_OUTPUT
		fAngleDeg	:	REAL;	(* Returns the clockwise rotation angle in degree *)
	END_VAR

END_FUNCTION

// Functions/Code Quality/F_VN_GradeQRCode

	{attribute 'TcIecLibraryType'}
	{attribute 'external_name' := 'F_VN_GradeQRCode_GUID_BC17E121_DBD0_BBA0_4E91_2886930332A8'}
	(* Grades a QR code according to ISO / IEC 15415:2011. Requires uniform illumination, good focus and the image sensor plane parallel to the code plane to achieve meaningful results. *)
	FUNCTION F_VN_GradeQRCode : HRESULT
	VAR_INPUT
		ipSrcImage	:	ITcVnImage;	(* Source image, only containing the QR code region (USINT, 1 channel, including quiet zone) *)
		ipDecodedData	:	REFERENCE TO ITcVnContainer;	(* Returns the decoded data (ContainerType_String_SINT) *)
	END_VAR
	VAR_IN_OUT
		stCodeGrades	:	TcVnCodeGradesQR;	(* Returns the code grades in the range from 0 (very bad) to 4 (very good) *)
	END_VAR
	VAR_INPUT
		fModuleWidth	:	REAL;	(* Minimum module width of the code in the image (in pixels). Must be at least 3, preferably 5 - 8. *)
		hrPrev	:	HRESULT;	(* HRESULT indicating the result of previous operations (If SUCCEEDED(hrPrev) equals false, no operation is executed.) *)
	END_VAR
	VAR_OUTPUT
		fAngleDeg	:	REAL;	(* Returns the clockwise rotation angle in degree *)
	END_VAR

END_FUNCTION

// Functions/Code Quality/F_VN_GradeQRCodeExp

	{attribute 'TcIecLibraryType'}
	{attribute 'external_name' := 'F_VN_GradeQRCodeExp_GUID_EF0F27E3_ACF2_BCB8_6190_C1A00B69652A'}
	(* Grades a QR code according to ISO / IEC 15415:2011. Requires uniform illumination, good focus and the image sensor plane parallel to the code plane to achieve meaningful results. (expert function) *)
	FUNCTION F_VN_GradeQRCodeExp : HRESULT
	VAR_INPUT
		ipSrcImage	:	ITcVnImage;	(* Source image, only containing the QR code region (USINT, 1 channel, including quiet zone) *)
		ipDecodedData	:	REFERENCE TO ITcVnContainer;	(* Returns the decoded data (ContainerType_String_SINT) *)
	END_VAR
	VAR_IN_OUT
		stCodeGrades	:	TcVnCodeGradesQR;	(* Returns the code grades in the range from 0 (very bad) to 4 (very good) *)
	END_VAR
	VAR_INPUT
		fModuleWidth	:	REAL;	(* Minimum module width of the code in the image (in pixels). Must be at least 3, preferably 5 - 8. *)
		ipResultVisualization	:	REFERENCE TO ITcVnImage;	(* Returns a visualization of the scan grid (optional, set to 0 if not required). Module margin grades are color coded: >= 3 as green, >= 2 as light blue, >= 1 as orange, < 1 as red *)
		ipMarginGrades	:	REFERENCE TO ITcVnContainer;	(* Returns the individual margin grade for each module, e.g. to create a custom visualization (optional, set to 0 if not required; ContainerType_Vector_TcVnVector3_REAL, containing [x-position, y-position, grade]) *)
		ipContour	:	REFERENCE TO ITcVnContainer;	(* Returns the 4 code corner points, excluding the quiet zone (optional, set to 0 if not required; ContainerType_Vector_TcVnPoint2_DINT) *)
		hrPrev	:	HRESULT;	(* HRESULT indicating the result of previous operations (If SUCCEEDED(hrPrev) equals false, no operation is executed.) *)
	END_VAR
	VAR_OUTPUT
		fAngleDeg	:	REAL;	(* Returns the clockwise rotation angle in degree *)
	END_VAR

END_FUNCTION

// Functions/Texture Analysis/F_VN_Granulometry

	{attribute 'TcIecLibraryType'}
	{attribute 'external_name' := 'F_VN_Granulometry_GUID_76CD1329_004A_B325_5AA4_1A824E70B520'}
	(* Computes the granulometry of a textured image using morphological operations. *)
	FUNCTION F_VN_Granulometry : HRESULT
	VAR_INPUT
		ipImage	:	ITcVnImage;	(* Source image (1 channel) *)
		ipIntensityDiffs	:	REFERENCE TO ITcVnContainer;	(* Returns the intensity differences between successive structuring element sizes (CTcVnContainer_Vector_LREAL), which can be used as features for texture description. *)
		eMorphType	:	ETcVnMorphologicalOperator;	(* Only opening or closing are supported. *)
		nMinSize	:	UDINT;	(* Min structuring element size (odd, >= 3) *)
		nMaxSize	:	UDINT;	(* Max structuring element size (>= nMinSize) *)
		nStep	:	UDINT;	(* Step, by which nMinSize is incremented until nMaxSize is exceeded (even, >= 2). *)
		hrPrev	:	HRESULT;	(* HRESULT indicating the result of previous operations (If SUCCEEDED(hrPrev) equals false, no operation is executed.) *)
	END_VAR

END_FUNCTION

// Functions/Texture Analysis/F_VN_HaralickFeatures

	{attribute 'TcIecLibraryType'}
	{attribute 'external_name' := 'F_VN_HaralickFeatures_GUID_5BCA76DF_787C_B4B7_7FB1_3D28B756E1E4'}
	(* Computes the Haralick features of a graylevel image, which describe the texture. *)
	FUNCTION F_VN_HaralickFeatures : HRESULT
	VAR_INPUT
		ipImage	:	ITcVnImage;	(* Source image (1 channel, USINT) *)
		ipFeatures	:	REFERENCE TO ITcVnContainer;	(* Returns the computed Haralick features (CTcVnContainer_Vector_LREAL). The returned feature set contains the mean and standard deviation for each of the first 13 Haralick features, computed for 0, 45, 90, 135 degrees. So there will be 26 features in total (f1 mean, f1 stdDev, f2 mean, f2 stdDev, ..., f13 mean, f13 stdDev). *)
		nDist	:	UDINT;	(* Distance *)
		hrPrev	:	HRESULT;	(* HRESULT indicating the result of previous operations (If SUCCEEDED(hrPrev) equals false, no operation is executed.) *)
	END_VAR

END_FUNCTION

// Functions/OCR/F_VN_OCR

	{attribute 'TcIecLibraryType'}
	{attribute 'external_name' := 'F_VN_OCR_GUID_DDC8991D_B2A9_B372_4096_C3F02F217550'}
	(* Detects and recognizes characters in a binary image (white characters on black background). *)
	FUNCTION F_VN_OCR : HRESULT
	VAR_INPUT
		ipSrcImage	:	ITcVnImage;	(* Source image (USINT, 1 channel, binary) *)
		eModel	:	ULINT;	(* Selection of OCR model types (ETcVnOcrModelType) *)
		ipCharacters	:	REFERENCE TO ITcVnContainer;	(* Returns the recognized characters (ContainerType_Vector_String_SINT) *)
		hrPrev	:	HRESULT;	(* HRESULT indicating the result of previous operations (If SUCCEEDED(hrPrev) equals false, no operation is executed.) *)
	END_VAR

END_FUNCTION

// Functions/OCR/F_VN_OCRExp

	{attribute 'TcIecLibraryType'}
	{attribute 'external_name' := 'F_VN_OCRExp_GUID_763DBE05_552C_B2A4_62BC_BE7FAD1FEEF4'}
	(* Detects and recognizes characters in a binary image (white characters on black background). (expert function) *)
	FUNCTION F_VN_OCRExp : HRESULT
	VAR_INPUT
		ipSrcImage	:	ITcVnImage;	(* Source image (USINT, 1 channel, binary) *)
		eModel	:	ULINT;	(* Selection of OCR model types (ETcVnOcrModelType) *)
		ipCharacters	:	REFERENCE TO ITcVnContainer;	(* Returns the recognized characters (ContainerType_Vector_String_SINT) *)
	END_VAR
	VAR_IN_OUT CONSTANT
		sPattern	:	STRING;	(* String pattern containing the format in which characters are presented *)
	END_VAR
	VAR_INPUT
		eOcrOptions	:	UDINT;	(* Specifies which options must be applied to the function (ETcVnOcrOptions) *)
		ipBoundingBoxes	:	REFERENCE TO ITcVnContainer;	(* Returns the corresponding bounding boxes of the recognized characters (ContainerType_Vector_TcVnRectangle_DINT, optional, set to 0 if not required) *)
		ipConfidences	:	REFERENCE TO ITcVnContainer;	(* Returns the corresponding classification confidences of the recognized characters (ContainerType_Vector_REAL, optional, set to 0 if not required) *)
		hrPrev	:	HRESULT;	(* HRESULT indicating the result of previous operations (If SUCCEEDED(hrPrev) equals false, no operation is executed.) *)
	END_VAR
	VAR_OUTPUT
		fMinConfidence	:	REAL;	(* Returns the minimum value of the confidences *)
	END_VAR

END_FUNCTION

// Functions/Code Reading/F_VN_ReadBarcode

	{attribute 'TcIecLibraryType'}
	{attribute 'external_name' := 'F_VN_ReadBarcode_GUID_16D4BA4F_6E1B_B966_6D00_89637101900D'}
	(* Detect and interpret a 1d barcode within the provided image.
          Can be canceled by Watchdog. *)
	FUNCTION F_VN_ReadBarcode : HRESULT
	VAR_INPUT
		ipSrcImage	:	ITcVnImage;	(* Source image (USINT elements, 1 channel or 3 channel (3 channel input is expected to be RGB and internally converted to Gray)) *)
		ipDecodedData	:	REFERENCE TO ITcVnContainer;	(* Returns the decoded code (ContainerType_Vector_String_SINT) *)
		eBarcodeType	:	UDINT;	(* Types of barcode to search for (ETcVnBarcodeType) *)
		hrPrev	:	HRESULT;	(* HRESULT indicating the result of previous operations (If SUCCEEDED(hrPrev) equals false, no operation is executed.) *)
	END_VAR

END_FUNCTION

// Functions/Code Reading/F_VN_ReadBarcodeExp

	{attribute 'TcIecLibraryType'}
	{attribute 'external_name' := 'F_VN_ReadBarcodeExp_GUID_1C5A2CF4_7F84_B35A_5FF5_42A55B70AEBE'}
	(* Detect and interpret a 1d barcode within the provided image.
          Can be canceled by Watchdog. *)
	FUNCTION F_VN_ReadBarcodeExp : HRESULT
	VAR_INPUT
		ipSrcImage	:	ITcVnImage;	(* Source image (USINT elements, 1 channel or 3 channel (3 channel input is expected to be RGB and internally converted to Gray)) *)
		ipDecodedData	:	REFERENCE TO ITcVnContainer;	(* Returns the decoded code (ContainerType_Vector_String_SINT) *)
		ipContours	:	REFERENCE TO ITcVnContainer;	(* Returns the code positions as contours (optional, set to 0 if not required; ContainerType_Vector_Vector_TcVnPoint2_DINT) *)
		eBarcodeType	:	UDINT;	(* Types of barcode to search for (ETcVnBarcodeType) *)
		nCodeNumber	:	DINT;	(* Number of 1d barcode that should be detected within the provided image (currently only 1 supported). *)
		eSearchDirection	:	ETcVnBarcodeSearchDirection;	(* Barcode search direction. *)
		hrPrev	:	HRESULT;	(* HRESULT indicating the result of previous operations (If SUCCEEDED(hrPrev) equals false, no operation is executed.) *)
	END_VAR

END_FUNCTION

// Functions/Code Reading/F_VN_ReadBarcodeExp2

	{attribute 'TcIecLibraryType'}
	{attribute 'external_name' := 'F_VN_ReadBarcodeExp2_GUID_DD996683_BB0D_B5A7_74CB_155BE8EEA769'}
	(* Detect and interpret a 1d barcode within the provided image.
          Can be canceled by Watchdog. *)
	FUNCTION F_VN_ReadBarcodeExp2 : HRESULT
	VAR_INPUT
		ipSrcImage	:	ITcVnImage;	(* Source image (USINT elements, 1 channel or 3 channel (3 channel input is expected to be RGB and internally converted to Gray)) *)
		ipDecodedData	:	REFERENCE TO ITcVnContainer;	(* Returns the decoded code (ContainerType_Vector_String_SINT) *)
		ipContours	:	REFERENCE TO ITcVnContainer;	(* Returns the code positions as contours (optional, set to 0 if not required; ContainerType_Vector_Vector_TcVnPoint2_DINT) *)
		eBarcodeType	:	UDINT;	(* Types of barcode to search for (ETcVnBarcodeType) *)
		nCodeNumber	:	DINT;	(* Number of 1d barcode that should be detected within the provided image (currently only 1 supported). *)
		eSearchDirection	:	ETcVnBarcodeSearchDirection;	(* Barcode search direction. *)
		ipAngles	:	REFERENCE TO ITcVnContainer;	(* Returns the clockwise code rotation angles (optional, set to 0 if not required; ContainerType_Vector_REAL) *)
		hrPrev	:	HRESULT;	(* HRESULT indicating the result of previous operations (If SUCCEEDED(hrPrev) equals false, no operation is executed.) *)
	END_VAR

END_FUNCTION

// Functions/Code Reading/F_VN_ReadDataMatrixCode

	{attribute 'TcIecLibraryType'}
	{attribute 'external_name' := 'F_VN_ReadDataMatrixCode_GUID_DC65A69C_8CF6_B172_4E79_F4413EAB75AE'}
	(* Detect and interpret a data matrix code (ECC200) within the provided image. *)
	FUNCTION F_VN_ReadDataMatrixCode : HRESULT
	VAR_INPUT
		ipSrcImage	:	ITcVnImage;	(* Source image (USINT elements, 1 or 3 channels) *)
		ipDecodedData	:	REFERENCE TO ITcVnContainer;	(* Returns the decoded code (ContainerType_Vector_String_SINT) *)
		hrPrev	:	HRESULT;	(* HRESULT indicating the result of previous operations (If SUCCEEDED(hrPrev) equals false, no operation is executed.) *)
	END_VAR

END_FUNCTION

// Functions/Code Reading/F_VN_ReadDataMatrixCodeExp

	{attribute 'TcIecLibraryType'}
	{attribute 'external_name' := 'F_VN_ReadDataMatrixCodeExp_GUID_423E565A_A43D_BE1B_6611_36532CD0B516'}
	(* Detect and interpret a data matrix code (ECC200) within the provided image. *)
	FUNCTION F_VN_ReadDataMatrixCodeExp : HRESULT
	VAR_INPUT
		ipSrcImage	:	ITcVnImage;	(* Source image (USINT elements, 1 or 3 channels) *)
		ipDecodedData	:	REFERENCE TO ITcVnContainer;	(* Returns the decoded code (ContainerType_Vector_String_SINT) *)
		ipContours	:	REFERENCE TO ITcVnContainer;	(* Returns the code positions as contours (optional, set to 0 if not required; ContainerType_Vector_Vector_TcVnPoint2_DINT) *)
		nCodeNumber	:	DINT;	(* Number of data matrix codes that should be detected within the provided image. (If set to -1, it tries to detect all data matrix codes.) *)
		eSearchStrategy	:	UDINT;	(* Used search strategy (ETcVn2dCodeSearchStrategy) *)
		hrPrev	:	HRESULT;	(* HRESULT indicating the result of previous operations (If SUCCEEDED(hrPrev) equals false, no operation is executed.) *)
	END_VAR

END_FUNCTION

// Functions/Code Reading/F_VN_ReadDataMatrixCodeExp2

	{attribute 'TcIecLibraryType'}
	{attribute 'external_name' := 'F_VN_ReadDataMatrixCodeExp2_GUID_92811DB6_0599_B3C6_6D15_352F37181069'}
	(* Detect and interpret a data matrix code (ECC200) within the provided image. *)
	FUNCTION F_VN_ReadDataMatrixCodeExp2 : HRESULT
	VAR_INPUT
		ipSrcImage	:	ITcVnImage;	(* Source image (USINT elements, 1 or 3 channels) *)
		ipDecodedData	:	REFERENCE TO ITcVnContainer;	(* Returns the decoded code (ContainerType_Vector_String_SINT) *)
		ipContours	:	REFERENCE TO ITcVnContainer;	(* Returns the code positions as contours (optional, set to 0 if not required; ContainerType_Vector_Vector_TcVnPoint2_DINT) *)
		nCodeNumber	:	DINT;	(* Number of data matrix codes that should be detected within the provided image. (If set to -1, it tries to detect all data matrix codes.) *)
		eSearchStrategy	:	UDINT;	(* Used search strategy (ETcVn2dCodeSearchStrategy) *)
		ipAngles	:	REFERENCE TO ITcVnContainer;	(* Returns the clockwise code rotation angles (optional, set to 0 if not required; ContainerType_Vector_REAL) *)
		hrPrev	:	HRESULT;	(* HRESULT indicating the result of previous operations (If SUCCEEDED(hrPrev) equals false, no operation is executed.) *)
	END_VAR

END_FUNCTION

// Functions/Code Reading/F_VN_ReadPharmaCode

	{attribute 'TcIecLibraryType'}
	{attribute 'external_name' := 'F_VN_ReadPharmaCode_GUID_8ED3E5A8_E91C_BCC0_685C_2CE28A311CFA'}
	(* Detect and interpret a pharma code within the provided image.
				Can be canceled by Watchdog. *)
	FUNCTION F_VN_ReadPharmaCode : HRESULT
	VAR_INPUT
		ipSrcImage	:	ITcVnImage;	(* Source image (1 channel (all element types) or 3 channel with elements of type TCVN_ET_USINT, TCVN_ET_UINT or TCVN_ET_REAL (3 channel input is expected to be RGB and internally converted to Gray)) *)
		ipDecodedData	:	REFERENCE TO ITcVnContainer;	(* Returns the decoded code (ContainerType_Vector_String_SINT) *)
		hrPrev	:	HRESULT;	(* HRESULT indicating the result of previous operations (If SUCCEEDED(hrPrev) equals false, no operation is executed.) *)
	END_VAR

END_FUNCTION

// Functions/Code Reading/F_VN_ReadPharmaCodeExp

	{attribute 'TcIecLibraryType'}
	{attribute 'external_name' := 'F_VN_ReadPharmaCodeExp_GUID_8BCDC08B_3068_BBC3_67E1_40F39D971AB1'}
	(* Detect and interpret a pharma code within the provided image.
				Can be canceled by Watchdog. *)
	FUNCTION F_VN_ReadPharmaCodeExp : HRESULT
	VAR_INPUT
		ipSrcImage	:	ITcVnImage;	(* Source image (1 channel (all element types) or 3 channel with elements of type TCVN_ET_USINT, TCVN_ET_UINT or TCVN_ET_REAL (3 channel input is expected to be RGB and internally converted to Gray)) *)
		ipDecodedData	:	REFERENCE TO ITcVnContainer;	(* Returns the decoded code (ContainerType_Vector_String_SINT) *)
		ipContours	:	REFERENCE TO ITcVnContainer;	(* Returns the code positions as contours (optional, set to 0 if not required; ContainerType_Vector_Vector_TcVnPoint2_DINT) *)
		nCodeNumber	:	DINT;	(* Number of pharma codes that should be detected within the provided image (currently only 1 supported). *)
		nMinBarNumber	:	INT;	(* Minimal number of (dark) bars that codes must have. *)
		hrPrev	:	HRESULT;	(* HRESULT indicating the result of previous operations (If SUCCEEDED(hrPrev) equals false, no operation is executed.) *)
	END_VAR

END_FUNCTION

// Functions/Code Reading/F_VN_ReadPharmaCodeExp2

	{attribute 'TcIecLibraryType'}
	{attribute 'external_name' := 'F_VN_ReadPharmaCodeExp2_GUID_0D01B133_51B8_B1CF_565E_F97419BE5CDF'}
	(* Detect and interpret a pharma code within the provided image.
				Can be canceled by Watchdog. *)
	FUNCTION F_VN_ReadPharmaCodeExp2 : HRESULT
	VAR_INPUT
		ipSrcImage	:	ITcVnImage;	(* Source image (1 channel (all element types) or 3 channel with elements of type TCVN_ET_USINT, TCVN_ET_UINT or TCVN_ET_REAL (3 channel input is expected to be RGB and internally converted to Gray)) *)
		ipDecodedData	:	REFERENCE TO ITcVnContainer;	(* Returns the decoded code (ContainerType_Vector_String_SINT) *)
		ipContours	:	REFERENCE TO ITcVnContainer;	(* Returns the code positions as contours (optional, set to 0 if not required; ContainerType_Vector_Vector_TcVnPoint2_DINT) *)
		nCodeNumber	:	DINT;	(* Number of pharma codes that should be detected within the provided image (currently only 1 supported). *)
		nMinBarNumber	:	INT;	(* Minimal number of (dark) bars that codes must have. *)
		ipAngles	:	REFERENCE TO ITcVnContainer;	(* Returns the clockwise code rotation angles (optional, set to 0 if not required; ContainerType_Vector_REAL) *)
		hrPrev	:	HRESULT;	(* HRESULT indicating the result of previous operations (If SUCCEEDED(hrPrev) equals false, no operation is executed.) *)
	END_VAR

END_FUNCTION

// Functions/Code Reading/F_VN_ReadQRCode

	{attribute 'TcIecLibraryType'}
	{attribute 'external_name' := 'F_VN_ReadQRCode_GUID_098C875D_FB34_B700_4386_FF8F89687138'}
	(* Detect and interpret a QR code within the provided image.
          Can be canceled by Watchdog. *)
	FUNCTION F_VN_ReadQRCode : HRESULT
	VAR_INPUT
		ipSrcImage	:	ITcVnImage;	(* Source image (USINT elements, 1 channel or 3 channel (3 channel input is expected to be RGB and internally converted to Gray)) *)
		ipDecodedData	:	REFERENCE TO ITcVnContainer;	(* Returns the decoded code (ContainerType_Vector_String_SINT) *)
		hrPrev	:	HRESULT;	(* HRESULT indicating the result of previous operations (If SUCCEEDED(hrPrev) equals false, no operation is executed.) *)
	END_VAR

END_FUNCTION

// Functions/Code Reading/F_VN_ReadQRCodeExp

	{attribute 'TcIecLibraryType'}
	{attribute 'external_name' := 'F_VN_ReadQRCodeExp_GUID_843C7CF8_E612_B139_48EB_A4590D84A86A'}
	(* Detect and interpret a QR code within the provided image.
          Can be canceled by Watchdog. *)
	FUNCTION F_VN_ReadQRCodeExp : HRESULT
	VAR_INPUT
		ipSrcImage	:	ITcVnImage;	(* Source image (USINT elements, 1 channel or 3 channel (3 channel input is expected to be RGB and internally converted to Gray)) *)
		ipDecodedData	:	REFERENCE TO ITcVnContainer;	(* Returns the decoded code (ContainerType_Vector_String_SINT) *)
		ipContours	:	REFERENCE TO ITcVnContainer;	(* Returns the code positions as contours (optional, set to 0 if not required; ContainerType_Vector_Vector_TcVnPoint2_DINT) *)
		nCodeNumber	:	DINT;	(* Number of QR codes that should be detected within the provided image (currently only 1 supported). *)
		eSearchStrategy	:	UDINT;	(* Used search strategy (ETcVn2dCodeSearchStrategy) *)
		hrPrev	:	HRESULT;	(* HRESULT indicating the result of previous operations (If SUCCEEDED(hrPrev) equals false, no operation is executed.) *)
	END_VAR

END_FUNCTION

// Functions/Code Reading/F_VN_ReadQRCodeExp2

	{attribute 'TcIecLibraryType'}
	{attribute 'external_name' := 'F_VN_ReadQRCodeExp2_GUID_A134283D_CC4A_BABF_74DE_99D7B8F80F30'}
	(* Detect and interpret a QR code within the provided image.
          Can be canceled by Watchdog. *)
	FUNCTION F_VN_ReadQRCodeExp2 : HRESULT
	VAR_INPUT
		ipSrcImage	:	ITcVnImage;	(* Source image (USINT elements, 1 channel or 3 channel (3 channel input is expected to be RGB and internally converted to Gray)) *)
		ipDecodedData	:	REFERENCE TO ITcVnContainer;	(* Returns the decoded code (ContainerType_Vector_String_SINT) *)
		ipContours	:	REFERENCE TO ITcVnContainer;	(* Returns the code positions as contours (optional, set to 0 if not required; ContainerType_Vector_Vector_TcVnPoint2_DINT) *)
		nCodeNumber	:	DINT;	(* Number of QR codes that should be detected within the provided image (currently only 1 supported). *)
		eSearchStrategy	:	UDINT;	(* Used search strategy (ETcVn2dCodeSearchStrategy) *)
		ipAngles	:	REFERENCE TO ITcVnContainer;	(* Returns the clockwise code rotation angles (optional, set to 0 if not required; ContainerType_Vector_REAL) *)
		hrPrev	:	HRESULT;	(* HRESULT indicating the result of previous operations (If SUCCEEDED(hrPrev) equals false, no operation is executed.) *)
	END_VAR

END_FUNCTION

// Functions/Algebraic Container Operations/F_VN_AddToContainerElements/F_VN_AddToContainerElements_DINT

	{attribute 'TcIecLibraryType'}
	{attribute 'external_name' := 'F_VN_AddToContainerElements_DINT_GUID_AFB2526B_F59F_B891_5913_263C77F748DC'}
	(* Add a value to each container element. *)
	FUNCTION F_VN_AddToContainerElements_DINT : HRESULT
	VAR_INPUT
		nValue	:	DINT;	(* Value *)
		ipContainer	:	ITcVnContainer;	(* Container with DINT elements *)
		hrPrev	:	HRESULT;	(* HRESULT indicating the result of previous operations (If SUCCEEDED(hrPrev) equals false, no operation is executed.) *)
	END_VAR

END_FUNCTION

// Functions/Algebraic Container Operations/F_VN_AddToContainerElements/F_VN_AddToContainerElements_INT

	{attribute 'TcIecLibraryType'}
	{attribute 'external_name' := 'F_VN_AddToContainerElements_INT_GUID_7247ABDE_FDC6_BA51_735E_97CE1A13F27A'}
	(* Add a value to each container element. *)
	FUNCTION F_VN_AddToContainerElements_INT : HRESULT
	VAR_INPUT
		nValue	:	INT;	(* Value *)
		ipContainer	:	ITcVnContainer;	(* Container with INT elements *)
		hrPrev	:	HRESULT;	(* HRESULT indicating the result of previous operations (If SUCCEEDED(hrPrev) equals false, no operation is executed.) *)
	END_VAR

END_FUNCTION

// Functions/Algebraic Container Operations/F_VN_AddToContainerElements/F_VN_AddToContainerElements_LREAL

	{attribute 'TcIecLibraryType'}
	{attribute 'external_name' := 'F_VN_AddToContainerElements_LREAL_GUID_103B982F_F52B_BEEA_60E8_FBF48F6EE950'}
	(* Add a value to each container element. *)
	FUNCTION F_VN_AddToContainerElements_LREAL : HRESULT
	VAR_INPUT
		fValue	:	LREAL;	(* Value *)
		ipContainer	:	ITcVnContainer;	(* Container with LREAL elements *)
		hrPrev	:	HRESULT;	(* HRESULT indicating the result of previous operations (If SUCCEEDED(hrPrev) equals false, no operation is executed.) *)
	END_VAR

END_FUNCTION

// Functions/Algebraic Container Operations/F_VN_AddToContainerElements/F_VN_AddToContainerElements_REAL

	{attribute 'TcIecLibraryType'}
	{attribute 'external_name' := 'F_VN_AddToContainerElements_REAL_GUID_9D0C37DB_9EEA_B4F7_718D_1E25A0453496'}
	(* Add a value to each container element. *)
	FUNCTION F_VN_AddToContainerElements_REAL : HRESULT
	VAR_INPUT
		fValue	:	REAL;	(* Value *)
		ipContainer	:	ITcVnContainer;	(* Container with REAL elements *)
		hrPrev	:	HRESULT;	(* HRESULT indicating the result of previous operations (If SUCCEEDED(hrPrev) equals false, no operation is executed.) *)
	END_VAR

END_FUNCTION

// Functions/Algebraic Container Operations/F_VN_AddToContainerElements/F_VN_AddToContainerElements_SINT

	{attribute 'TcIecLibraryType'}
	{attribute 'external_name' := 'F_VN_AddToContainerElements_SINT_GUID_D64EB219_A436_B0E3_73BF_79A1245B647E'}
	(* Add a value to each container element. *)
	FUNCTION F_VN_AddToContainerElements_SINT : HRESULT
	VAR_INPUT
		nValue	:	SINT;	(* Value *)
		ipContainer	:	ITcVnContainer;	(* Container with SINT elements *)
		hrPrev	:	HRESULT;	(* HRESULT indicating the result of previous operations (If SUCCEEDED(hrPrev) equals false, no operation is executed.) *)
	END_VAR

END_FUNCTION

// Functions/Algebraic Container Operations/F_VN_AddToContainerElements/F_VN_AddToContainerElements_TcVnKeyPoint

	{attribute 'TcIecLibraryType'}
	{attribute 'external_name' := 'F_VN_AddToContainerElements_TcVnKeyPoint_GUID_CF7E3264_9632_B05A_5E50_E3F35D849356'}
	(* Add a value to each container element. *)
	FUNCTION F_VN_AddToContainerElements_TcVnKeyPoint : HRESULT
	VAR_IN_OUT
		stValue	:	TcVnKeyPoint;	(* Value *)
	END_VAR
	VAR_INPUT
		ipContainer	:	ITcVnContainer;	(* Container with TcVnKeyPoint elements *)
		hrPrev	:	HRESULT;	(* HRESULT indicating the result of previous operations (If SUCCEEDED(hrPrev) equals false, no operation is executed.) *)
	END_VAR

END_FUNCTION

// Functions/Algebraic Container Operations/F_VN_AddToContainerElements/F_VN_AddToContainerElements_TcVnPoint2_DINT

	{attribute 'TcIecLibraryType'}
	{attribute 'external_name' := 'F_VN_AddToContainerElements_TcVnPoint2_DINT_GUID_F5A23A27_157C_B307_6CF9_F8D1F575BC20'}
	(* Add a value to each container element. *)
	FUNCTION F_VN_AddToContainerElements_TcVnPoint2_DINT : HRESULT
	VAR_IN_OUT
		aValue	:	TcVnPoint2_DINT;	(* Value *)
	END_VAR
	VAR_INPUT
		ipContainer	:	ITcVnContainer;	(* Container with TcVnPoint2_DINT elements *)
		hrPrev	:	HRESULT;	(* HRESULT indicating the result of previous operations (If SUCCEEDED(hrPrev) equals false, no operation is executed.) *)
	END_VAR

END_FUNCTION

// Functions/Algebraic Container Operations/F_VN_AddToContainerElements/F_VN_AddToContainerElements_TcVnPoint2_LREAL

	{attribute 'TcIecLibraryType'}
	{attribute 'external_name' := 'F_VN_AddToContainerElements_TcVnPoint2_LREAL_GUID_B751626B_1C87_B0DC_52A5_67E9B45F87FB'}
	(* Add a value to each container element. *)
	FUNCTION F_VN_AddToContainerElements_TcVnPoint2_LREAL : HRESULT
	VAR_IN_OUT
		aValue	:	TcVnPoint2_LREAL;	(* Value *)
	END_VAR
	VAR_INPUT
		ipContainer	:	ITcVnContainer;	(* Container with TcVnPoint2_LREAL elements *)
		hrPrev	:	HRESULT;	(* HRESULT indicating the result of previous operations (If SUCCEEDED(hrPrev) equals false, no operation is executed.) *)
	END_VAR

END_FUNCTION

// Functions/Algebraic Container Operations/F_VN_AddToContainerElements/F_VN_AddToContainerElements_TcVnPoint2_REAL

	{attribute 'TcIecLibraryType'}
	{attribute 'external_name' := 'F_VN_AddToContainerElements_TcVnPoint2_REAL_GUID_F4B12E31_AC5A_B321_65BE_779C18F7FF2F'}
	(* Add a value to each container element. *)
	FUNCTION F_VN_AddToContainerElements_TcVnPoint2_REAL : HRESULT
	VAR_IN_OUT
		aValue	:	TcVnPoint2_REAL;	(* Value *)
	END_VAR
	VAR_INPUT
		ipContainer	:	ITcVnContainer;	(* Container with TcVnPoint2_REAL elements *)
		hrPrev	:	HRESULT;	(* HRESULT indicating the result of previous operations (If SUCCEEDED(hrPrev) equals false, no operation is executed.) *)
	END_VAR

END_FUNCTION

// Functions/Algebraic Container Operations/F_VN_AddToContainerElements/F_VN_AddToContainerElements_TcVnPoint3_LREAL

	{attribute 'TcIecLibraryType'}
	{attribute 'external_name' := 'F_VN_AddToContainerElements_TcVnPoint3_LREAL_GUID_77BCD440_CEE2_BF2C_4759_935DB01A7128'}
	(* Add a value to each container element. *)
	FUNCTION F_VN_AddToContainerElements_TcVnPoint3_LREAL : HRESULT
	VAR_IN_OUT
		aValue	:	TcVnPoint3_LREAL;	(* Value *)
	END_VAR
	VAR_INPUT
		ipContainer	:	ITcVnContainer;	(* Container with TcVnPoint3_LREAL elements *)
		hrPrev	:	HRESULT;	(* HRESULT indicating the result of previous operations (If SUCCEEDED(hrPrev) equals false, no operation is executed.) *)
	END_VAR

END_FUNCTION

// Functions/Algebraic Container Operations/F_VN_AddToContainerElements/F_VN_AddToContainerElements_TcVnPoint3_REAL

	{attribute 'TcIecLibraryType'}
	{attribute 'external_name' := 'F_VN_AddToContainerElements_TcVnPoint3_REAL_GUID_8BA11F2F_E268_BD21_713F_FF70D11DB965'}
	(* Add a value to each container element. *)
	FUNCTION F_VN_AddToContainerElements_TcVnPoint3_REAL : HRESULT
	VAR_IN_OUT
		aValue	:	TcVnPoint3_REAL;	(* Value *)
	END_VAR
	VAR_INPUT
		ipContainer	:	ITcVnContainer;	(* Container with TcVnPoint3_REAL elements *)
		hrPrev	:	HRESULT;	(* HRESULT indicating the result of previous operations (If SUCCEEDED(hrPrev) equals false, no operation is executed.) *)
	END_VAR

END_FUNCTION

// Functions/Algebraic Container Operations/F_VN_AddToContainerElements/F_VN_AddToContainerElements_TcVnRectangle_DINT

	{attribute 'TcIecLibraryType'}
	{attribute 'external_name' := 'F_VN_AddToContainerElements_TcVnRectangle_DINT_GUID_A37399D3_FE09_BCD8_7895_3CE432EC6CC1'}
	(* Add a value to each container element. *)
	FUNCTION F_VN_AddToContainerElements_TcVnRectangle_DINT : HRESULT
	VAR_IN_OUT
		stValue	:	TcVnRectangle_DINT;	(* Value *)
	END_VAR
	VAR_INPUT
		ipContainer	:	ITcVnContainer;	(* Container with TcVnRectangle_DINT elements *)
		hrPrev	:	HRESULT;	(* HRESULT indicating the result of previous operations (If SUCCEEDED(hrPrev) equals false, no operation is executed.) *)
	END_VAR

END_FUNCTION

// Functions/Algebraic Container Operations/F_VN_AddToContainerElements/F_VN_AddToContainerElements_TcVnVector2_DINT

	{attribute 'TcIecLibraryType'}
	{attribute 'external_name' := 'F_VN_AddToContainerElements_TcVnVector2_DINT_GUID_09245AED_056B_B88A_51D1_35E2F458AC75'}
	(* Add a value to each container element. *)
	FUNCTION F_VN_AddToContainerElements_TcVnVector2_DINT : HRESULT
	VAR_IN_OUT
		aValue	:	TcVnVector2_DINT;	(* Value *)
	END_VAR
	VAR_INPUT
		ipContainer	:	ITcVnContainer;	(* Container with TcVnVector2_DINT elements *)
		hrPrev	:	HRESULT;	(* HRESULT indicating the result of previous operations (If SUCCEEDED(hrPrev) equals false, no operation is executed.) *)
	END_VAR

END_FUNCTION

// Functions/Algebraic Container Operations/F_VN_AddToContainerElements/F_VN_AddToContainerElements_TcVnVector2_INT

	{attribute 'TcIecLibraryType'}
	{attribute 'external_name' := 'F_VN_AddToContainerElements_TcVnVector2_INT_GUID_AE5820DD_81B9_B6EF_791A_0F801E8CB7A8'}
	(* Add a value to each container element. *)
	FUNCTION F_VN_AddToContainerElements_TcVnVector2_INT : HRESULT
	VAR_IN_OUT
		aValue	:	TcVnVector2_INT;	(* Value *)
	END_VAR
	VAR_INPUT
		ipContainer	:	ITcVnContainer;	(* Container with TcVnVector2_INT elements *)
		hrPrev	:	HRESULT;	(* HRESULT indicating the result of previous operations (If SUCCEEDED(hrPrev) equals false, no operation is executed.) *)
	END_VAR

END_FUNCTION

// Functions/Algebraic Container Operations/F_VN_AddToContainerElements/F_VN_AddToContainerElements_TcVnVector2_REAL

	{attribute 'TcIecLibraryType'}
	{attribute 'external_name' := 'F_VN_AddToContainerElements_TcVnVector2_REAL_GUID_EC512B39_17F0_B42E_6949_96413C6B5013'}
	(* Add a value to each container element. *)
	FUNCTION F_VN_AddToContainerElements_TcVnVector2_REAL : HRESULT
	VAR_IN_OUT
		aValue	:	TcVnVector2_REAL;	(* Value *)
	END_VAR
	VAR_INPUT
		ipContainer	:	ITcVnContainer;	(* Container with TcVnVector2_REAL elements *)
		hrPrev	:	HRESULT;	(* HRESULT indicating the result of previous operations (If SUCCEEDED(hrPrev) equals false, no operation is executed.) *)
	END_VAR

END_FUNCTION

// Functions/Algebraic Container Operations/F_VN_AddToContainerElements/F_VN_AddToContainerElements_TcVnVector2_SINT

	{attribute 'TcIecLibraryType'}
	{attribute 'external_name' := 'F_VN_AddToContainerElements_TcVnVector2_SINT_GUID_4EA7CBFD_423E_BA63_43C8_E6874366D8BF'}
	(* Add a value to each container element. *)
	FUNCTION F_VN_AddToContainerElements_TcVnVector2_SINT : HRESULT
	VAR_IN_OUT
		aValue	:	TcVnVector2_SINT;	(* Value *)
	END_VAR
	VAR_INPUT
		ipContainer	:	ITcVnContainer;	(* Container with TcVnVector2_SINT elements *)
		hrPrev	:	HRESULT;	(* HRESULT indicating the result of previous operations (If SUCCEEDED(hrPrev) equals false, no operation is executed.) *)
	END_VAR

END_FUNCTION

// Functions/Algebraic Container Operations/F_VN_AddToContainerElements/F_VN_AddToContainerElements_TcVnVector2_UINT

	{attribute 'TcIecLibraryType'}
	{attribute 'external_name' := 'F_VN_AddToContainerElements_TcVnVector2_UINT_GUID_A2143006_AFFF_BE8E_6B65_506958A7FF58'}
	(* Add a value to each container element. *)
	FUNCTION F_VN_AddToContainerElements_TcVnVector2_UINT : HRESULT
	VAR_IN_OUT
		aValue	:	TcVnVector2_UINT;	(* Value *)
	END_VAR
	VAR_INPUT
		ipContainer	:	ITcVnContainer;	(* Container with TcVnVector2_UINT elements *)
		hrPrev	:	HRESULT;	(* HRESULT indicating the result of previous operations (If SUCCEEDED(hrPrev) equals false, no operation is executed.) *)
	END_VAR

END_FUNCTION

// Functions/Algebraic Container Operations/F_VN_AddToContainerElements/F_VN_AddToContainerElements_TcVnVector2_USINT

	{attribute 'TcIecLibraryType'}
	{attribute 'external_name' := 'F_VN_AddToContainerElements_TcVnVector2_USINT_GUID_EDA1F340_8D87_BC06_762E_73CF301C5FAB'}
	(* Add a value to each container element. *)
	FUNCTION F_VN_AddToContainerElements_TcVnVector2_USINT : HRESULT
	VAR_IN_OUT
		aValue	:	TcVnVector2_USINT;	(* Value *)
	END_VAR
	VAR_INPUT
		ipContainer	:	ITcVnContainer;	(* Container with TcVnVector2_USINT elements *)
		hrPrev	:	HRESULT;	(* HRESULT indicating the result of previous operations (If SUCCEEDED(hrPrev) equals false, no operation is executed.) *)
	END_VAR

END_FUNCTION

// Functions/Algebraic Container Operations/F_VN_AddToContainerElements/F_VN_AddToContainerElements_TcVnVector3_INT

	{attribute 'TcIecLibraryType'}
	{attribute 'external_name' := 'F_VN_AddToContainerElements_TcVnVector3_INT_GUID_85FD7A91_8C08_BF15_756A_7A9B0320B75B'}
	(* Add a value to each container element. *)
	FUNCTION F_VN_AddToContainerElements_TcVnVector3_INT : HRESULT
	VAR_IN_OUT
		aValue	:	TcVnVector3_INT;	(* Value *)
	END_VAR
	VAR_INPUT
		ipContainer	:	ITcVnContainer;	(* Container with TcVnVector3_INT elements *)
		hrPrev	:	HRESULT;	(* HRESULT indicating the result of previous operations (If SUCCEEDED(hrPrev) equals false, no operation is executed.) *)
	END_VAR

END_FUNCTION

// Functions/Algebraic Container Operations/F_VN_AddToContainerElements/F_VN_AddToContainerElements_TcVnVector3_REAL

	{attribute 'TcIecLibraryType'}
	{attribute 'external_name' := 'F_VN_AddToContainerElements_TcVnVector3_REAL_GUID_F38F496C_03FE_B4E7_6009_F2FE7BCEDE65'}
	(* Add a value to each container element. *)
	FUNCTION F_VN_AddToContainerElements_TcVnVector3_REAL : HRESULT
	VAR_IN_OUT
		aValue	:	TcVnVector3_REAL;	(* Value *)
	END_VAR
	VAR_INPUT
		ipContainer	:	ITcVnContainer;	(* Container with TcVnVector3_REAL elements *)
		hrPrev	:	HRESULT;	(* HRESULT indicating the result of previous operations (If SUCCEEDED(hrPrev) equals false, no operation is executed.) *)
	END_VAR

END_FUNCTION

// Functions/Algebraic Container Operations/F_VN_AddToContainerElements/F_VN_AddToContainerElements_TcVnVector3_SINT

	{attribute 'TcIecLibraryType'}
	{attribute 'external_name' := 'F_VN_AddToContainerElements_TcVnVector3_SINT_GUID_9F7EF153_9EF5_B4F4_5AE3_CB687256CAFB'}
	(* Add a value to each container element. *)
	FUNCTION F_VN_AddToContainerElements_TcVnVector3_SINT : HRESULT
	VAR_IN_OUT
		aValue	:	TcVnVector3_SINT;	(* Value *)
	END_VAR
	VAR_INPUT
		ipContainer	:	ITcVnContainer;	(* Container with TcVnVector3_SINT elements *)
		hrPrev	:	HRESULT;	(* HRESULT indicating the result of previous operations (If SUCCEEDED(hrPrev) equals false, no operation is executed.) *)
	END_VAR

END_FUNCTION

// Functions/Algebraic Container Operations/F_VN_AddToContainerElements/F_VN_AddToContainerElements_TcVnVector3_UINT

	{attribute 'TcIecLibraryType'}
	{attribute 'external_name' := 'F_VN_AddToContainerElements_TcVnVector3_UINT_GUID_361B23D6_BBD8_BE16_6DCC_9C4FBE18FCCE'}
	(* Add a value to each container element. *)
	FUNCTION F_VN_AddToContainerElements_TcVnVector3_UINT : HRESULT
	VAR_IN_OUT
		aValue	:	TcVnVector3_UINT;	(* Value *)
	END_VAR
	VAR_INPUT
		ipContainer	:	ITcVnContainer;	(* Container with TcVnVector3_UINT elements *)
		hrPrev	:	HRESULT;	(* HRESULT indicating the result of previous operations (If SUCCEEDED(hrPrev) equals false, no operation is executed.) *)
	END_VAR

END_FUNCTION

// Functions/Algebraic Container Operations/F_VN_AddToContainerElements/F_VN_AddToContainerElements_TcVnVector3_USINT

	{attribute 'TcIecLibraryType'}
	{attribute 'external_name' := 'F_VN_AddToContainerElements_TcVnVector3_USINT_GUID_23731CFD_7F79_B242_6A58_43D67949960C'}
	(* Add a value to each container element. *)
	FUNCTION F_VN_AddToContainerElements_TcVnVector3_USINT : HRESULT
	VAR_IN_OUT
		aValue	:	TcVnVector3_USINT;	(* Value *)
	END_VAR
	VAR_INPUT
		ipContainer	:	ITcVnContainer;	(* Container with TcVnVector3_USINT elements *)
		hrPrev	:	HRESULT;	(* HRESULT indicating the result of previous operations (If SUCCEEDED(hrPrev) equals false, no operation is executed.) *)
	END_VAR

END_FUNCTION

// Functions/Algebraic Container Operations/F_VN_AddToContainerElements/F_VN_AddToContainerElements_TcVnVector4_DINT

	{attribute 'TcIecLibraryType'}
	{attribute 'external_name' := 'F_VN_AddToContainerElements_TcVnVector4_DINT_GUID_2363C7E1_7FF4_BCA1_743D_4B556CCE4DE5'}
	(* Add a value to each container element. *)
	FUNCTION F_VN_AddToContainerElements_TcVnVector4_DINT : HRESULT
	VAR_IN_OUT
		aValue	:	TcVnVector4_DINT;	(* Value *)
	END_VAR
	VAR_INPUT
		ipContainer	:	ITcVnContainer;	(* Container with TcVnVector4_DINT elements *)
		hrPrev	:	HRESULT;	(* HRESULT indicating the result of previous operations (If SUCCEEDED(hrPrev) equals false, no operation is executed.) *)
	END_VAR

END_FUNCTION

// Functions/Algebraic Container Operations/F_VN_AddToContainerElements/F_VN_AddToContainerElements_TcVnVector4_INT

	{attribute 'TcIecLibraryType'}
	{attribute 'external_name' := 'F_VN_AddToContainerElements_TcVnVector4_INT_GUID_A3A21D35_2633_B0B9_73C7_4F843085CCBE'}
	(* Add a value to each container element. *)
	FUNCTION F_VN_AddToContainerElements_TcVnVector4_INT : HRESULT
	VAR_IN_OUT
		aValue	:	TcVnVector4_INT;	(* Value *)
	END_VAR
	VAR_INPUT
		ipContainer	:	ITcVnContainer;	(* Container with TcVnVector4_INT elements *)
		hrPrev	:	HRESULT;	(* HRESULT indicating the result of previous operations (If SUCCEEDED(hrPrev) equals false, no operation is executed.) *)
	END_VAR

END_FUNCTION

// Functions/Algebraic Container Operations/F_VN_AddToContainerElements/F_VN_AddToContainerElements_TcVnVector4_LREAL

	{attribute 'TcIecLibraryType'}
	{attribute 'external_name' := 'F_VN_AddToContainerElements_TcVnVector4_LREAL_GUID_C224188D_04D3_B465_4967_A3469E288B86'}
	(* Add a value to each container element. *)
	FUNCTION F_VN_AddToContainerElements_TcVnVector4_LREAL : HRESULT
	VAR_IN_OUT
		aValue	:	TcVnVector4_LREAL;	(* Value *)
	END_VAR
	VAR_INPUT
		ipContainer	:	ITcVnContainer;	(* Container with TcVnVector4_LREAL elements *)
		hrPrev	:	HRESULT;	(* HRESULT indicating the result of previous operations (If SUCCEEDED(hrPrev) equals false, no operation is executed.) *)
	END_VAR

END_FUNCTION

// Functions/Algebraic Container Operations/F_VN_AddToContainerElements/F_VN_AddToContainerElements_TcVnVector4_SINT

	{attribute 'TcIecLibraryType'}
	{attribute 'external_name' := 'F_VN_AddToContainerElements_TcVnVector4_SINT_GUID_EC01C8DA_F0D6_BEF5_4E8D_5B1485F6A432'}
	(* Add a value to each container element. *)
	FUNCTION F_VN_AddToContainerElements_TcVnVector4_SINT : HRESULT
	VAR_IN_OUT
		aValue	:	TcVnVector4_SINT;	(* Value *)
	END_VAR
	VAR_INPUT
		ipContainer	:	ITcVnContainer;	(* Container with TcVnVector4_SINT elements *)
		hrPrev	:	HRESULT;	(* HRESULT indicating the result of previous operations (If SUCCEEDED(hrPrev) equals false, no operation is executed.) *)
	END_VAR

END_FUNCTION

// Functions/Algebraic Container Operations/F_VN_AddToContainerElements/F_VN_AddToContainerElements_TcVnVector4_UINT

	{attribute 'TcIecLibraryType'}
	{attribute 'external_name' := 'F_VN_AddToContainerElements_TcVnVector4_UINT_GUID_A5A6D6C5_E691_BEFC_44EE_3CB7A7417459'}
	(* Add a value to each container element. *)
	FUNCTION F_VN_AddToContainerElements_TcVnVector4_UINT : HRESULT
	VAR_IN_OUT
		aValue	:	TcVnVector4_UINT;	(* Value *)
	END_VAR
	VAR_INPUT
		ipContainer	:	ITcVnContainer;	(* Container with TcVnVector4_UINT elements *)
		hrPrev	:	HRESULT;	(* HRESULT indicating the result of previous operations (If SUCCEEDED(hrPrev) equals false, no operation is executed.) *)
	END_VAR

END_FUNCTION

// Functions/Algebraic Container Operations/F_VN_AddToContainerElements/F_VN_AddToContainerElements_TcVnVector4_USINT

	{attribute 'TcIecLibraryType'}
	{attribute 'external_name' := 'F_VN_AddToContainerElements_TcVnVector4_USINT_GUID_837974F0_4C77_B74E_70E0_B890B1BAE31E'}
	(* Add a value to each container element. *)
	FUNCTION F_VN_AddToContainerElements_TcVnVector4_USINT : HRESULT
	VAR_IN_OUT
		aValue	:	TcVnVector4_USINT;	(* Value *)
	END_VAR
	VAR_INPUT
		ipContainer	:	ITcVnContainer;	(* Container with TcVnVector4_USINT elements *)
		hrPrev	:	HRESULT;	(* HRESULT indicating the result of previous operations (If SUCCEEDED(hrPrev) equals false, no operation is executed.) *)
	END_VAR

END_FUNCTION

// Functions/Algebraic Container Operations/F_VN_AddToContainerElements/F_VN_AddToContainerElements_UDINT

	{attribute 'TcIecLibraryType'}
	{attribute 'external_name' := 'F_VN_AddToContainerElements_UDINT_GUID_AAEC2BB0_82A0_BD07_5EBB_E1BA9731394D'}
	(* Add a value to each container element. *)
	FUNCTION F_VN_AddToContainerElements_UDINT : HRESULT
	VAR_INPUT
		nValue	:	UDINT;	(* Value *)
		ipContainer	:	ITcVnContainer;	(* Container with UDINT elements *)
		hrPrev	:	HRESULT;	(* HRESULT indicating the result of previous operations (If SUCCEEDED(hrPrev) equals false, no operation is executed.) *)
	END_VAR

END_FUNCTION

// Functions/Algebraic Container Operations/F_VN_AddToContainerElements/F_VN_AddToContainerElements_UINT

	{attribute 'TcIecLibraryType'}
	{attribute 'external_name' := 'F_VN_AddToContainerElements_UINT_GUID_5EE8B6B3_A8DD_B83B_6D9A_AEB5ED33B191'}
	(* Add a value to each container element. *)
	FUNCTION F_VN_AddToContainerElements_UINT : HRESULT
	VAR_INPUT
		nValue	:	UINT;	(* Value *)
		ipContainer	:	ITcVnContainer;	(* Container with UINT elements *)
		hrPrev	:	HRESULT;	(* HRESULT indicating the result of previous operations (If SUCCEEDED(hrPrev) equals false, no operation is executed.) *)
	END_VAR

END_FUNCTION

// Functions/Algebraic Container Operations/F_VN_AddToContainerElements/F_VN_AddToContainerElements_ULINT

	{attribute 'TcIecLibraryType'}
	{attribute 'external_name' := 'F_VN_AddToContainerElements_ULINT_GUID_719E92AC_182A_B1C7_5D1A_894B9AAA29EC'}
	(* Add a value to each container element. *)
	FUNCTION F_VN_AddToContainerElements_ULINT : HRESULT
	VAR_INPUT
		nValue	:	ULINT;	(* Value *)
		ipContainer	:	ITcVnContainer;	(* Container with ULINT elements *)
		hrPrev	:	HRESULT;	(* HRESULT indicating the result of previous operations (If SUCCEEDED(hrPrev) equals false, no operation is executed.) *)
	END_VAR

END_FUNCTION

// Functions/Algebraic Container Operations/F_VN_AddToContainerElements/F_VN_AddToContainerElements_USINT

	{attribute 'TcIecLibraryType'}
	{attribute 'external_name' := 'F_VN_AddToContainerElements_USINT_GUID_AFD29392_7750_BF31_77BA_C2CC2E98500B'}
	(* Add a value to each container element. *)
	FUNCTION F_VN_AddToContainerElements_USINT : HRESULT
	VAR_INPUT
		nValue	:	USINT;	(* Value *)
		ipContainer	:	ITcVnContainer;	(* Container with USINT elements *)
		hrPrev	:	HRESULT;	(* HRESULT indicating the result of previous operations (If SUCCEEDED(hrPrev) equals false, no operation is executed.) *)
	END_VAR

END_FUNCTION

// Functions/Image Analysis/Object Detection/F_VN_AdjustActiveContour

	{attribute 'TcIecLibraryType'}
	{attribute 'external_name' := 'F_VN_AdjustActiveContour_GUID_1C8942FC_0080_B77A_78EF_2A5FB9402731'}
	(* Adjust active contour (snake) in order to minimize its cummulative (internal and external) energy. *)
	FUNCTION F_VN_AdjustActiveContour : HRESULT
	VAR_INPUT
		ipImage	:	ITcVnImage;	(* Source image (1 channel, USINT elements) *)
		ipActiveContour	:	ITcVnContainer;	(* Initial contour, which will be adjusted *)
		fAlpha	:	REAL;	(* Continuity energy coefficient *)
		fBeta	:	REAL;	(* Curvature energy coefficient *)
		fGamma	:	REAL;	(* Image energy coefficient *)
		nWindowWidth	:	UDINT;	(* Window width (3, 5, 7, ...) *)
		nWindowHeight	:	UDINT;	(* Window height (3, 5, 7, ...) *)
		nMaxIterations	:	UDINT;	(* Maximum iterations *)
		bUseGradient	:	BOOL;	(* If true, the gradient magnitude is used as image energy (otherwise: pixel intensity) *)
		hrPrev	:	HRESULT;	(* HRESULT indicating the result of previous operations (If SUCCEEDED(hrPrev) equals false, no operation is executed.) *)
	END_VAR

END_FUNCTION

// Functions/Image Analysis/Object Detection/F_VN_DetectBlobs

	{attribute 'TcIecLibraryType'}
	{attribute 'external_name' := 'F_VN_DetectBlobs_GUID_2D4AF51B_6AF3_B7F3_45ED_FCED45AF4E58'}
	(* Detects blob-contours. Applies a threshold, a contour search and offers several options for filtering the found contours. Provides easy setup for multiple thresholds and combination of results. *)
	FUNCTION F_VN_DetectBlobs : HRESULT
	VAR_INPUT
		ipSrcImage	:	ITcVnImage;	(* Source image (USINT or REAL, 1 channel or 3 channel (3 channel input is expected to be RGB and internally converted to Gray)) *)
		ipBlobContours	:	REFERENCE TO ITcVnContainer;	(* Returns a container which is filled with the found contours (ContainerType_Vector_Vector_TcVnPoint2_DINT; The elements of this container are single contours. Non-zero interface pointers are reused.) *)
	END_VAR
	VAR_IN_OUT
		stParams	:	TcVnParamsBlobDetection;	(* Parameters to filter the detected contours. *)
	END_VAR
	VAR_INPUT
		hrPrev	:	HRESULT;	(* HRESULT indicating the result of previous operations (If SUCCEEDED(hrPrev) equals false, no operation is executed.) *)
	END_VAR

END_FUNCTION

// Functions/Image Analysis/Object Detection/F_VN_DetectBlobsExp

	{attribute 'TcIecLibraryType'}
	{attribute 'external_name' := 'F_VN_DetectBlobsExp_GUID_08305532_BC98_B763_6F5A_2C434AA43CF2'}
	(* Detects blob-contours. Applies a threshold, a contour search and offers several options for filtering the found contours. Provides easy setup for multiple thresholds and combination of results. (expert function) *)
	FUNCTION F_VN_DetectBlobsExp : HRESULT
	VAR_INPUT
		ipSrcImage	:	ITcVnImage;	(* Source image (USINT or REAL, 1 channel or 3 channel (3 channel input is expected to be RGB and internally converted to Gray)) *)
		ipBlobContours	:	REFERENCE TO ITcVnContainer;	(* Returns a container which is filled with the found contours (ContainerType_Vector_Vector_TcVnPoint2_DINT; The elements of this container are single contours. Non-zero interface pointers are reused.) *)
	END_VAR
	VAR_IN_OUT
		stParams	:	TcVnParamsBlobDetection;	(* Parameters to filter the detected contours. *)
		aOffset	:	TcVnPoint;	(* Offset by which every contour point is shifted *)
	END_VAR
	VAR_INPUT
		hrPrev	:	HRESULT;	(* HRESULT indicating the result of previous operations (If SUCCEEDED(hrPrev) equals false, no operation is executed.) *)
	END_VAR

END_FUNCTION

// Functions/Image Analysis/Object Detection/F_VN_FindContourHierarchyExp

	{attribute 'TcIecLibraryType'}
	{attribute 'external_name' := 'F_VN_FindContourHierarchyExp_GUID_6052C7B8_AD42_B4BE_6AD4_BBB56579CA70'}
	(* Search for object contours in a binary image and determine their hierarchical relationship. (expert function) *)
	FUNCTION F_VN_FindContourHierarchyExp : HRESULT
	VAR_INPUT
		ipSrcImage	:	ITcVnImage;	(* Source image (1 channel, binary) *)
		ipContours	:	REFERENCE TO ITcVnContainer;	(* Returns a container which is filled with the found contours (ContainerType_Vector_Vector_TcVnPoint2_DINT; The elements of this container are single contours. Non-zero interface pointers are reused.) *)
		ipHierarchy	:	REFERENCE TO ITcVnContainer;	(* Returns a container which is filled with information on the found contours' hierarchy (ContainerType_Vector_TcVnVector4_DINT; The elements of this container are four-dimensional vectors containing the 0-based indices of the next [0] and the previous contour [1] at the same level, the first child [2], and the parent [3]. Non-zero interface pointers are reused.) *)
		eRetrievalMode	:	ETcVnContourRetrievalMode;	(* Specifies which contours are retrieved and how their relationship is encoded *)
		eApproximationMethod	:	ETcVnContourApproximationMethod;	(* Contour encoding *)
	END_VAR
	VAR_IN_OUT
		aOffset	:	TcVnPoint;	(* Offset by which every contour point is shifted *)
	END_VAR
	VAR_INPUT
		hrPrev	:	HRESULT;	(* HRESULT indicating the result of previous operations (If SUCCEEDED(hrPrev) equals false, no operation is executed.) *)
	END_VAR

END_FUNCTION

// Functions/Image Analysis/Object Detection/F_VN_FindContours

	{attribute 'TcIecLibraryType'}
	{attribute 'external_name' := 'F_VN_FindContours_GUID_0899EACF_1ABE_B78D_5C4F_13F17D863083'}
	(* Search for object contours in a binary image. Returns only external contours. *)
	FUNCTION F_VN_FindContours : HRESULT
	VAR_INPUT
		ipSrcImage	:	ITcVnImage;	(* Source image (1 channel, binary) *)
		ipContours	:	REFERENCE TO ITcVnContainer;	(* Returns a container which is filled with the found contours (ContainerType_Vector_Vector_TcVnPoint2_DINT; The elements of this container are single contours. Non-zero interface pointers are reused.) *)
		hrPrev	:	HRESULT;	(* HRESULT indicating the result of previous operations (If SUCCEEDED(hrPrev) equals false, no operation is executed.) *)
	END_VAR

END_FUNCTION

// Functions/Image Analysis/Object Detection/F_VN_FindContoursExp

	{attribute 'TcIecLibraryType'}
	{attribute 'external_name' := 'F_VN_FindContoursExp_GUID_789B2953_71E4_B59B_7854_ED69F0F908ED'}
	(* Search for object contours in a binary image. (expert function) *)
	FUNCTION F_VN_FindContoursExp : HRESULT
	VAR_INPUT
		ipSrcImage	:	ITcVnImage;	(* Source image (1 channel, binary) *)
		ipContours	:	REFERENCE TO ITcVnContainer;	(* Returns a container which is filled with the found contours (ContainerType_Vector_Vector_TcVnPoint2_DINT; The elements of this container are single contours. Non-zero interface pointers are reused.) *)
		eRetrievalMode	:	ETcVnContourRetrievalMode;	(* Specifies which contours are retrieved and how their relationship is encoded *)
		eApproximationMethod	:	ETcVnContourApproximationMethod;	(* Contour encoding *)
	END_VAR
	VAR_IN_OUT
		aOffset	:	TcVnPoint;	(* Offset by which every contour point is shifted *)
	END_VAR
	VAR_INPUT
		hrPrev	:	HRESULT;	(* HRESULT indicating the result of previous operations (If SUCCEEDED(hrPrev) equals false, no operation is executed.) *)
	END_VAR

END_FUNCTION

// Functions/Image Analysis/Object Detection/F_VN_HoughCircles

